KUKA KRL program: MyProgram_036().src

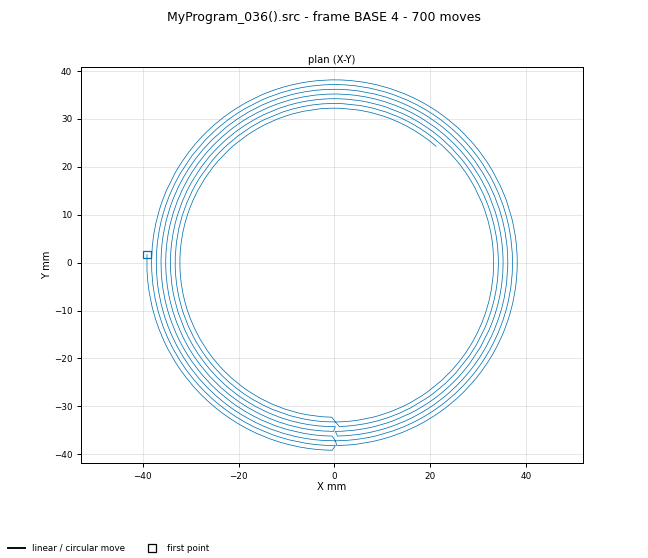
[picture p0: tool path of MyProgram_036().src in frame BASE 4, 700 of 700 moves have a stored position in this frame; points joined in program order, loops and branches not executed]
&ACCESS RVP
&REL 1
&PARAM TEMPLATE = C:\KRC\Roboter\Template\vorgabe
&PARAM EDITMASK = *
DEF MyProgram_036()
; ---- Setting reference (Base) ----
$BASE = BASE_DATA[4]

; --------------------------
; ---- Setting tool (TCP) ----
$TOOL = TOOL_DATA[3]
; --------------------------

$VEL.CP = VEL_APROX_PRINT
Startdeposition()
$VEL.CP = VEL_PRINT
LIN {X -39.1246,Y 1.7119,Z 61,A 171.6311,B 24.8459,C -2.8635,E1 24.8398,E2 -448.4299} C_DIS
LIN {X -39.1359,Y -1.4401,Z 61,A 176.0807,B 24.8477,C -2.8474,E1 24.84,E2 -452.8678} C_DIS
LIN {X -38.9837,Y -3.7356,Z 61,A 179.6269,B 24.8486,C -2.8388,E1 24.8408,E2 -456.4147} C_DIS
LIN {X -38.6887,Y -6.0708,Z 61,A -176.4142,B 24.8492,C -2.8336,E1 24.8424,E2 -460.3847} C_DIS
LIN {X -38.045,Y -9.2867,Z 61,A -172.1524,B 24.8513,C -2.8136,E1 24.8449,E2 -464.6237} C_DIS
LIN {X -37.3515,Y -11.7707,Z 61,A -167.9795,B 24.852,C -2.8066,E1 24.8483,E2 -468.8041} C_DIS
LIN {X -36.6288,Y -13.8562,Z 61,A -164.8858,B 24.8532,C -2.796,E1 24.8512,E2 -471.8898} C_DIS
LIN {X -35.5913,Y -16.3387,Z 61,A -160.9363,B 24.8543,C -2.7852,E1 24.8557,E2 -475.8352} C_DIS
LIN {X -34.7861,Y -17.9895,Z 61,A -158.0445,B 24.8548,C -2.7801,E1 24.8594,E2 -478.7304} C_DIS
LIN {X -33.1861,Y -20.7929,Z 61,A -154.2853,B 24.8572,C -2.7576,E1 24.8646,E2 -482.4552} C_DIS
LIN {X -32.2724,Y -22.1845,Z 61,A -151.2973,B 24.8572,C -2.7576,E1 24.8693,E2 -485.4579} C_DIS
LIN {X -31.1359,Y -23.754,Z 61,A -148.272,B 24.8577,C -2.7529,E1 24.8744,E2 -488.4866} C_DIS
LIN {X -29.5277,Y -25.725,Z 61,A -144.6978,B 24.8587,C -2.7428,E1 24.8808,E2 -492.0533} C_DIS
LIN {X -28.1922,Y -27.182,Z 61,A -141.5616,B 24.8591,C -2.7394,E1 24.8868,E2 -495.1951} C_DIS
LIN {X -26.3524,Y -28.9697,Z 61,A -138.0117,B 24.8601,C -2.7297,E1 24.894,E2 -498.7362} C_DIS
LIN {X -24.7345,Y -30.3624,Z 61,A -135.1218,B 24.8609,C -2.7212,E1 24.9001,E2 -501.617} C_DIS
LIN {X -23.6269,Y -31.2322,Z 61,A -132.7128,B 24.8609,C -2.7217,E1 24.9055,E2 -504.036} C_DIS
LIN {X -21.8691,Y -32.4872,Z 61,A -129.5903,B 24.8614,C -2.7162,E1 24.9127,E2 -507.1559} C_DIS
LIN {X -20.1827,Y -33.5602,Z 61,A -126.7285,B 24.8619,C -2.7112,E1 24.9195,E2 -510.0148} C_DIS
LIN {X -18.2564,Y -34.6463,Z 61,A -123.3846,B 24.8622,C -2.7083,E1 24.9277,E2 -513.3613} C_DIS
LIN {X -16.2163,Y -35.6471,Z 61,A -119.632,B 24.8621,C -2.7099,E1 24.9372,E2 -517.127} C_DIS
LIN {X -13.4921,Y -36.7645,Z 61,A -115.8847,B 24.8632,C -2.6989,E1 24.9469,E2 -520.856} C_DIS
LIN {X -11.6052,Y -37.4029,Z 61,A -112.8226,B 24.8632,C -2.6986,E1 24.955,E2 -523.9229} C_DIS
LIN {X -9.5171,Y -37.9887,Z 61,A -109.6569,B 24.8634,C -2.6966,E1 24.9636,E2 -527.0887} C_DIS
LIN {X -7.0999,Y -38.5133,Z 61,A -106.0841,B 24.8636,C -2.6946,E1 24.9733,E2 -530.6608} C_DIS
LIN {X -5.4376,Y -38.7827,Z 61,A -103.9005,B 24.8641,C -2.6903,E1 24.9794,E2 -532.8361} C_DIS
LIN {X -3.7877,Y -38.9789,Z 61,A -101.2031,B 24.8638,C -2.6936,E1 24.9869,E2 -535.5429} C_DIS
LIN {X -2.1489,Y -39.103,Z 61,A -99.0333,B 24.8641,C -2.6905,E1 24.9929,E2 -537.7062} C_DIS
LIN {X -0.4519,Y -39.16,Z 61,A -96.2889,B 24.8637,C -2.6944,E1 25.0006,E2 -540.4601} C_DIS
LIN {X -0.4519,Y -39.16,Z 61,A -96.2889,B 24.8637,C -2.6944,E1 25.0006,E2 -540.4601} C_DIS
Enddeposition()
LIN {X 0.2058,Y -38.174,Z 61,A -96.4617,B 24.8635,C -2.6964,E1 25.0001,E2 -540.2922} C_DIS
Startdeposition()
$VEL.CP = VEL_PRINT
LIN {X -1.6251,Y -38.1424,Z 61,A -99.5524,B 24.864,C -2.6916,E1 24.9915,E2 -537.1895} C_DIS
LIN {X -3.7981,Y -37.9874,Z 61,A -103.2763,B 24.8645,C -2.686,E1 24.9811,E2 -533.4505} C_DIS
LIN {X -5.7354,Y -37.7438,Z 61,A -106.8998,B 24.8653,C -2.6781,E1 24.971,E2 -529.8052} C_DIS
LIN {X -9.3911,Y -37.0041,Z 61,A -111.3776,B 24.8637,C -2.6944,E1 24.9589,E2 -525.3603} C_DIS
LIN {X -11.7237,Y -36.3323,Z 61,A -114.7703,B 24.8631,C -2.6999,E1 24.9498,E2 -521.975} C_DIS
LIN {X -12.9207,Y -35.9244,Z 61,A -117.5141,B 24.864,C -2.6915,E1 24.9426,E2 -519.2057} C_DIS
LIN {X -16.5245,Y -34.4154,Z 61,A -122.843,B 24.8627,C -2.7039,E1 24.929,E2 -513.8936} C_DIS
LIN {X -18.8039,Y -33.2249,Z 61,A -126.9062,B 24.8624,C -2.7066,E1 24.919,E2 -509.8253} C_DIS
LIN {X -20.5168,Y -32.1953,Z 61,A -129.5033,B 24.8615,C -2.7154,E1 24.9129,E2 -507.2414} C_DIS
LIN {X -21.5761,Y -31.496,Z 61,A -131.5541,B 24.8614,C -2.7168,E1 24.9081,E2 -505.1869} C_DIS
LIN {X -22.9175,Y -30.5331,Z 61,A -134.0934,B 24.861,C -2.7203,E1 24.9024,E2 -502.647} C_DIS
LIN {X -24.5041,Y -29.2754,Z 61,A -136.9789,B 24.8603,C -2.7274,E1 24.8962,E2 -499.7676} C_DIS
LIN {X -25.6498,Y -28.2775,Z 61,A -139.37,B 24.86,C -2.7306,E1 24.8912,E2 -497.3745} C_DIS
LIN {X -26.978,Y -27.0123,Z 61,A -142.0686,B 24.8593,C -2.7367,E1 24.8858,E2 -494.6794} C_DIS
LIN {X -28.1489,Y -25.79,Z 61,A -144.6778,B 24.8588,C -2.7414,E1 24.8808,E2 -492.07} C_DIS
LIN {X -29.33,Y -24.4382,Z 61,A -147.3487,B 24.8582,C -2.7477,E1 24.876,E2 -489.4019} C_DIS
LIN {X -30.4284,Y -23.0568,Z 61,A -149.8973,B 24.8575,C -2.7549,E1 24.8716,E2 -486.8585} C_DIS
LIN {X -31.2137,Y -21.9816,Z 61,A -152.4219,B 24.8575,C -2.7544,E1 24.8675,E2 -484.3202} C_DIS
LIN {X -32.4672,Y -20.0846,Z 61,A -155.857,B 24.8566,C -2.7627,E1 24.8623,E2 -480.8877} C_DIS
LIN {X -33.8432,Y -17.6674,Z 61,A -159.701,B 24.8551,C -2.777,E1 24.8572,E2 -477.0576} C_DIS
LIN {X -34.9349,Y -15.3963,Z 61,A -163.7856,B 24.8544,C -2.7844,E1 24.8524,E2 -472.9685} C_DIS
LIN {X -35.7598,Y -13.369,Z 61,A -167.3157,B 24.8536,C -2.7914,E1 24.8488,E2 -469.4352} C_DIS
LIN {X -36.7499,Y -10.3404,Z 61,A -171.6234,B 24.8517,C -2.81,E1 24.8453,E2 -465.1472} C_DIS
LIN {X -37.4441,Y -7.4482,Z 61,A -177.1229,B 24.8513,C -2.8136,E1 24.842,E2 -459.6239} C_DIS
LIN {X -37.8937,Y -4.6464,Z 61,A 179.0092,B 24.8495,C -2.8303,E1 24.8406,E2 -455.7729} C_DIS
LIN {X -38.1362,Y -1.7679,Z 61,A 175.1413,B 24.8476,C -2.8482,E1 24.8399,E2 -451.9246} C_DIS
LIN {X -38.1731,Y 0.5611,Z 61,A 170.9288,B 24.8471,C -2.8524,E1 24.8399,E2 -447.6968} C_DIS
LIN {X -38.0202,Y 3.4564,Z 61,A 167.0952,B 24.8451,C -2.8709,E1 24.8407,E2 -443.8844} C_DIS
LIN {X -37.7315,Y 5.815,Z 61,A 163.5178,B 24.844,C -2.8819,E1 24.842,E2 -440.3121} C_DIS
LIN {X -37.28,Y 8.2277,Z 61,A 159.4344,B 24.8431,C -2.8896,E1 24.8444,E2 -436.2229} C_DIS
LIN {X -36.5358,Y 11.0755,Z 61,A 155.6693,B 24.841,C -2.9093,E1 24.8472,E2 -432.4832} C_DIS
LIN {X -35.9396,Y 12.8788,Z 61,A 152.4915,B 24.8404,C -2.9148,E1 24.85,E2 -429.3004} C_DIS
LIN {X -35.1002,Y 15.0163,Z 61,A 148.4463,B 24.8399,C -2.9193,E1 24.8544,E2 -425.2436} C_DIS
LIN {X -33.2218,Y 18.8107,Z 61,A 143.1464,B 24.8367,C -2.9477,E1 24.8611,E2 -419.9833} C_DIS
LIN {X -32.099,Y 20.6674,Z 61,A 138.9421,B 24.8367,C -2.9475,E1 24.8674,E2 -415.757} C_DIS
LIN {X -30.4008,Y 23.0936,Z 61,A 134.5485,B 24.8354,C -2.9597,E1 24.8746,E2 -411.3713} C_DIS
LIN {X -28.9431,Y 24.896,Z 61,A 131.6927,B 24.8337,C -2.9747,E1 24.8797,E2 -408.5383} C_DIS
LIN {X -27.8474,Y 26.1152,Z 61,A 129.0954,B 24.8332,C -2.9793,E1 24.8846,E2 -405.9406} C_DIS
LIN {X -26.5489,Y 27.4343,Z 61,A 126.228,B 24.8326,C -2.9849,E1 24.8902,E2 -403.0744} C_DIS
LIN {X -24.9689,Y 28.8796,Z 61,A 122.2932,B 24.8326,C -2.9846,E1 24.8985,E2 -399.1234} C_DIS
LIN {X -22.971,Y 30.4929,Z 61,A 119.3529,B 24.8306,C -3.0021,E1 24.9049,E2 -396.2141} C_DIS
LIN {X -20.951,Y 31.9146,Z 61,A 114.7776,B 24.8308,C -3,E1 24.9155,E2 -391.6186} C_DIS
LIN {X -18.3987,Y 33.4508,Z 61,A 110.4355,B 24.8298,C -3.0091,E1 24.9261,E2 -387.2853} C_DIS
LIN {X -15.4253,Y 34.9224,Z 61,A 106.0547,B 24.8282,C -3.0232,E1 24.937,E2 -382.9271} C_DIS
LIN {X -13.9822,Y 35.5244,Z 61,A 103.7511,B 24.8278,C -3.0269,E1 24.943,E2 -380.6271} C_DIS
LIN {X -12.4032,Y 36.1066,Z 61,A 101.0674,B 24.8276,C -3.0282,E1 24.9501,E2 -377.9413} C_DIS
LIN {X -10.6068,Y 36.6745,Z 61,A 98.1852,B 24.8274,C -3.0307,E1 24.9578,E2 -375.06} C_DIS
LIN {X -8.7748,Y 37.1544,Z 61,A 94.9865,B 24.8275,C -3.0292,E1 24.9665,E2 -371.8533} C_DIS
LIN {X -6.2361,Y 37.6642,Z 61,A 91.3939,B 24.8268,C -3.0356,E1 24.9763,E2 -368.2722} C_DIS
LIN {X -3.4721,Y 38.0188,Z 61,A 86.7795,B 24.8271,C -3.0326,E1 24.9891,E2 -363.648} C_DIS
LIN {X -0.5874,Y 38.1726,Z 61,A 82.9526,B 24.8263,C -3.0402,E1 24.9997,E2 -359.8384} C_DIS
LIN {X 1.5062,Y 38.1473,Z 61,A 79.9793,B 24.826,C -3.0427,E1 25.008,E2 -356.8715} C_DIS
LIN {X 3.3481,Y 38.03,Z 61,A 76.4399,B 24.8271,C -3.0328,E1 25.0179,E2 -353.3105} C_DIS
LIN {X 6.3001,Y 37.6535,Z 61,A 72.8307,B 24.826,C -3.0427,E1 25.0278,E2 -349.728} C_DIS
LIN {X 8.7875,Y 37.1523,Z 61,A 68.6153,B 24.8268,C -3.0356,E1 25.0394,E2 -345.5011} C_DIS
LIN {X 11.5673,Y 36.3827,Z 61,A 63.6954,B 24.828,C -3.0247,E1 25.0526,E2 -340.564} C_DIS
LIN {X 14.6024,Y 35.2747,Z 61,A 59.3124,B 24.8278,C -3.0264,E1 25.064,E2 -336.1945} C_DIS
LIN {X 16.5716,Y 34.3928,Z 61,A 56.4111,B 24.8278,C -3.0273,E1 25.0713,E2 -333.3029} C_DIS
LIN {X 18.0246,Y 33.6545,Z 61,A 54.01,B 24.828,C -3.0248,E1 25.0772,E2 -330.9025} C_DIS
LIN {X 19.4873,Y 32.8288,Z 61,A 51.7271,B 24.828,C -3.0247,E1 25.0827,E2 -328.6262} C_DIS
LIN {X 20.561,Y 32.1673,Z 61,A 49.7273,B 24.8285,C -3.0203,E1 25.0875,E2 -326.6224} C_DIS
LIN {X 21.7389,Y 31.3832,Z 61,A 47.3022,B 24.8294,C -3.0126,E1 25.0931,E2 -324.1873} C_DIS
LIN {X 23.4845,Y 30.0999,Z 61,A 43.8809,B 24.8303,C -3.0045,E1 25.1007,E2 -320.7592} C_DIS
LIN {X 25.6796,Y 28.2502,Z 61,A 40.0705,B 24.8304,C -3.0036,E1 25.1087,E2 -316.9615} C_DIS
LIN {X 26.6253,Y 27.3604,Z 61,A 37.5195,B 24.8319,C -2.9908,E1 25.1139,E2 -314.3909} C_DIS
LIN {X 28.6369,Y 25.2476,Z 61,A 33.4573,B 24.8324,C -2.986,E1 25.1215,E2 -310.3351} C_DIS
LIN {X 30.1948,Y 23.3613,Z 61,A 29.8375,B 24.8333,C -2.9783,E1 25.1279,E2 -306.7139} C_DIS
LIN {X 31.7933,Y 21.1349,Z 61,A 25.3674,B 24.835,C -2.9628,E1 25.135,E2 -302.229} C_DIS
LIN {X 32.9335,Y 19.3101,Z 61,A 22.073,B 24.8361,C -2.9534,E1 25.1397,E2 -298.9294} C_DIS
LIN {X 34.6066,Y 16.1204,Z 61,A 17.177,B 24.8368,C -2.9466,E1 25.1458,E2 -294.0434} C_DIS
LIN {X 35.5024,Y 14.0382,Z 61,A 13.9544,B 24.8376,C -2.9399,E1 25.1493,E2 -290.8225} C_DIS
LIN {X 35.9963,Y 12.7183,Z 61,A 11.2382,B 24.8393,C -2.9244,E1 25.1518,E2 -288.085} C_DIS
LIN {X 37.0311,Y 9.2859,Z 61,A 6.2712,B 24.8403,C -2.915,E1 25.1556,E2 -283.124} C_DIS
LIN {X 37.3917,Y 7.7034,Z 61,A 3.9387,B 24.841,C -2.9092,E1 25.1569,E2 -280.7916} C_DIS
LIN {X 37.7634,Y 5.6075,Z 61,A 0.7109,B 24.8421,C -2.8989,E1 25.1584,E2 -277.5584} C_DIS
LIN {X 37.9807,Y 3.8676,Z 61,A -1.8164,B 24.8428,C -2.8925,E1 25.1592,E2 -275.0307} C_DIS
LIN {X 38.1283,Y 1.9349,Z 61,A -4.6115,B 24.8436,C -2.8852,E1 25.1597,E2 -272.235} C_DIS
LIN {X 38.1752,Y 0.4157,Z 61,A -6.7829,B 24.8442,C -2.8798,E1 25.1597,E2 -270.0638} C_DIS
LIN {X 38.1514,Y -1.4106,Z 61,A -9.8132,B 24.8456,C -2.8666,E1 25.1596,E2 -267.0204} C_DIS
LIN {X 38.0292,Y -3.3592,Z 61,A -12.4507,B 24.8461,C -2.8621,E1 25.159,E2 -264.3877} C_DIS
LIN {X 37.7783,Y -5.5026,Z 61,A -15.9673,B 24.8477,C -2.8475,E1 25.1577,E2 -260.8574} C_DIS
LIN {X 37.249,Y -8.3648,Z 61,A -20.7885,B 24.8499,C -2.8268,E1 25.155,E2 -256.0153} C_DIS
LIN {X 36.6348,Y -10.7419,Z 61,A -23.6115,B 24.8496,C -2.8291,E1 25.1529,E2 -253.2138} C_DIS
LIN {X 36.227,Y -12.0447,Z 61,A -25.7983,B 24.8505,C -2.8206,E1 25.151,E2 -251.0194} C_DIS
LIN {X 35.4552,Y -14.1583,Z 61,A -28.9661,B 24.8513,C -2.8138,E1 25.1479,E2 -247.8531} C_DIS
LIN {X 34.7913,Y -15.7177,Z 61,A -31.8323,B 24.8526,C -2.8012,E1 25.1447,E2 -244.9727} C_DIS
LIN {X 33.868,Y -17.6204,Z 61,A -34.7421,B 24.8531,C -2.7961,E1 25.141,E2 -242.0665} C_DIS
LIN {X 33.0339,Y -19.1379,Z 61,A -37.4369,B 24.8541,C -2.7872,E1 25.1373,E2 -239.3646} C_DIS
LIN {X 32.2579,Y -20.4193,Z 61,A -40.0322,B 24.8553,C -2.7756,E1 25.1334,E2 -236.755} C_DIS
LIN {X 30.6847,Y -22.715,Z 61,A -43.7394,B 24.8557,C -2.7717,E1 25.1275,E2 -233.0564} C_DIS
LIN {X 29.6057,Y -24.1037,Z 61,A -46.2431,B 24.8562,C -2.7669,E1 25.1231,E2 -230.5532} C_DIS
LIN {X 28.6953,Y -25.1808,Z 61,A -48.7794,B 24.8574,C -2.7552,E1 25.1185,E2 -228.0005} C_DIS
LIN {X 26.8749,Y -27.1148,Z 61,A -52.4982,B 24.858,C -2.7496,E1 25.1112,E2 -224.2846} C_DIS
LIN {X 25.4921,Y -28.4183,Z 61,A -55.5822,B 24.859,C -2.7396,E1 25.1049,E2 -221.1894} C_DIS
LIN {X 23.4955,Y -30.091,Z 61,A -59.0641,B 24.8592,C -2.7376,E1 25.0974,E2 -217.7159} C_DIS
LIN {X 22.3346,Y -30.9625,Z 61,A -61.3187,B 24.8598,C -2.732,E1 25.0923,E2 -215.4561} C_DIS
LIN {X 20.9688,Y -31.9029,Z 61,A -64.0449,B 24.8607,C -2.7237,E1 25.0859,E2 -212.7194} C_DIS
LIN {X 18.8062,Y -33.2233,Z 61,A -67.5439,B 24.8609,C -2.7213,E1 25.0775,E2 -209.2255} C_DIS
LIN {X 17.0992,Y -34.1339,Z 61,A -70.8441,B 24.862,C -2.7109,E1 25.0693,E2 -205.9096} C_DIS
LIN {X 14.4634,Y -35.3313,Z 61,A -75.3242,B 24.8628,C -2.7027,E1 25.0578,E2 -201.4207} C_DIS
LIN {X 11.9187,Y -36.2692,Z 61,A -78.7995,B 24.8625,C -2.7059,E1 25.0487,E2 -197.9601} C_DIS
LIN {X 9.9784,Y -36.8499,Z 61,A -82.0849,B 24.8632,C -2.6992,E1 25.0398,E2 -194.6643} C_DIS
LIN {X 7.9305,Y -37.3437,Z 61,A -85.4763,B 24.8638,C -2.6932,E1 25.0306,E2 -191.2633} C_DIS
LIN {X 4.7796,Y -37.8768,Z 61,A -89.56,B 24.8632,C -2.6994,E1 25.0194,E2 -187.1982} C_DIS
LIN {X 2.7394,Y -38.0789,Z 61,A -93.3905,B 24.8643,C -2.6879,E1 25.0086,E2 -183.3425} C_DIS
LIN {X 0.4929,Y -38.1744,Z 61,A -96.4487,B 24.864,C -2.6909,E1 25.0001,E2 -180.2922} C_DIS
LIN {X 0.4929,Y -38.1744,Z 61,A -96.4487,B 24.864,C -2.6909,E1 25.0001,E2 -180.2922} C_DIS
Enddeposition()
LIN {X 0.2169,Y -37.1885,Z 61,A -97.0627,B 24.8625,C -2.7057,E1 24.9985,E2 -179.7131} C_DIS
Startdeposition()
$VEL.CP = VEL_PRINT
LIN {X 2.3849,Y -37.1156,Z 61,A -91.3777,B 24.8593,C -2.7372,E1 25.0146,E2 -185.4716} C_DIS
LIN {X 4.4565,Y -36.9242,Z 61,A -88.3914,B 24.8593,C -2.7362,E1 25.0228,E2 -188.4532} C_DIS
LIN {X 7.033,Y -36.5207,Z 61,A -84.9258,B 24.8598,C -2.7317,E1 25.0323,E2 -191.9046} C_DIS
LIN {X 8.6705,Y -36.1675,Z 61,A -81.6512,B 24.8586,C -2.7437,E1 25.0413,E2 -195.203} C_DIS
LIN {X 12.3086,Y -35.0962,Z 61,A -76.6912,B 24.8592,C -2.7381,E1 25.0544,E2 -200.1407} C_DIS
LIN {X 14.4746,Y -34.2597,Z 61,A -72.4913,B 24.8578,C -2.7518,E1 25.0654,E2 -204.3637} C_DIS
LIN {X 16.5626,Y -33.3005,Z 61,A -69.4009,B 24.8578,C -2.7509,E1 25.0731,E2 -207.4438} C_DIS
LIN {X 18.2017,Y -32.4337,Z 61,A -66.4981,B 24.8573,C -2.7564,E1 25.0803,E2 -210.3514} C_DIS
LIN {X 19.8235,Y -31.4689,Z 61,A -63.5956,B 24.8567,C -2.7617,E1 25.0872,E2 -213.2571} C_DIS
LIN {X 21.6468,Y -30.2433,Z 61,A -60.2084,B 24.856,C -2.7684,E1 25.095,E2 -216.6487} C_DIS
LIN {X 23.1585,Y -29.1023,Z 61,A -57.1197,B 24.8551,C -2.777,E1 25.1018,E2 -219.7466} C_DIS
LIN {X 25.1549,Y -27.3948,Z 61,A -53.3687,B 24.8547,C -2.7817,E1 25.1096,E2 -223.4936} C_DIS
LIN {X 26.8232,Y -25.7636,Z 61,A -49.4807,B 24.8533,C -2.7947,E1 25.1173,E2 -227.3959} C_DIS
LIN {X 28.2812,Y -24.154,Z 61,A -46.3833,B 24.8528,C -2.7992,E1 25.123,E2 -230.4902} C_DIS
LIN {X 29.3197,Y -22.8833,Z 61,A -44.0555,B 24.8524,C -2.8027,E1 25.1271,E2 -232.8153} C_DIS
LIN {X 30.3514,Y -21.4954,Z 61,A -41.1551,B 24.8513,C -2.8135,E1 25.1318,E2 -235.7271} C_DIS
LIN {X 31.3778,Y -19.9674,Z 61,A -38.5235,B 24.8508,C -2.8181,E1 25.1359,E2 -238.3565} C_DIS
LIN {X 32.3405,Y -18.3676,Z 61,A -35.4557,B 24.8496,C -2.8291,E1 25.1402,E2 -241.4347} C_DIS
LIN {X 33.2135,Y -16.7376,Z 61,A -32.7932,B 24.8491,C -2.8344,E1 25.1436,E2 -244.0957} C_DIS
LIN {X 34.1529,Y -14.7256,Z 61,A -29.1477,B 24.8476,C -2.8481,E1 25.1478,E2 -247.7536} C_DIS
LIN {X 35.1839,Y -12.0569,Z 61,A -24.4656,B 24.8457,C -2.8657,E1 25.1523,E2 -252.4513} C_DIS
LIN {X 35.8338,Y -9.9607,Z 61,A -21.81,B 24.8458,C -2.8646,E1 25.1544,E2 -255.089} C_DIS
LIN {X 36.3501,Y -7.8679,Z 61,A -18.0003,B 24.8439,C -2.8826,E1 25.1568,E2 -258.9194} C_DIS
LIN {X 36.86,Y -4.9553,Z 61,A -13.15,B 24.8418,C -2.9016,E1 25.1588,E2 -263.786} C_DIS
LIN {X 37.1169,Y -2.3657,Z 61,A -9.6045,B 24.8412,C -2.9067,E1 25.1596,E2 -267.3227} C_DIS
LIN {X 37.1908,Y -0.1047,Z 61,A -6.4021,B 24.8405,C -2.9132,E1 25.1598,E2 -270.5213} C_DIS
LIN {X 37.1307,Y 2.1343,Z 61,A -2.5235,B 24.8386,C -2.9307,E1 25.1593,E2 -274.4183} C_DIS
LIN {X 36.8227,Y 5.2278,Z 61,A 2.0615,B 24.8373,C -2.9422,E1 25.1578,E2 -279.0035} C_DIS
LIN {X 36.3889,Y 7.6901,Z 61,A 5.9718,B 24.8359,C -2.9548,E1 25.1557,E2 -282.9208} C_DIS
LIN {X 35.9015,Y 9.7122,Z 61,A 9.0106,B 24.8351,C -2.9618,E1 25.1536,E2 -285.9585} C_DIS
LIN {X 35.2316,Y 11.9155,Z 61,A 12.6038,B 24.8339,C -2.9728,E1 25.1505,E2 -289.5575} C_DIS
LIN {X 34.2434,Y 14.5133,Z 61,A 16.4426,B 24.8333,C -2.9781,E1 25.1466,E2 -293.3875} C_DIS
LIN {X 33.3854,Y 16.3914,Z 61,A 19.7505,B 24.8321,C -2.9888,E1 25.1426,E2 -296.7028} C_DIS
LIN {X 32.6017,Y 17.8994,Z 61,A 22.5447,B 24.831,C -2.9984,E1 25.1389,E2 -299.5052} C_DIS
LIN {X 31.0625,Y 20.454,Z 61,A 27.4269,B 24.8292,C -3.0145,E1 25.1316,E2 -304.4009} C_DIS
LIN {X 29.9798,Y 22.0103,Z 61,A 30.226,B 24.8286,C -3.0197,E1 25.1271,E2 -307.1988} C_DIS
LIN {X 28.5043,Y 23.8906,Z 61,A 33.4788,B 24.8284,C -3.0217,E1 25.1213,E2 -310.4413} C_DIS
LIN {X 27.2141,Y 25.3508,Z 61,A 36.673,B 24.8273,C -3.0311,E1 25.1153,E2 -313.6436} C_DIS
LIN {X 25.9716,Y 26.6224,Z 61,A 39.0983,B 24.8272,C -3.0322,E1 25.1106,E2 -316.0611} C_DIS
LIN {X 24.9231,Y 27.6063,Z 61,A 41.2999,B 24.8267,C -3.0364,E1 25.106,E2 -318.2637} C_DIS
LIN {X 23.5916,Y 28.7528,Z 61,A 44.243,B 24.8257,C -3.0448,E1 25.0997,E2 -321.2155} C_DIS
LIN {X 22.1541,Y 29.8745,Z 61,A 46.8689,B 24.8255,C -3.047,E1 25.0939,E2 -323.8372} C_DIS
LIN {X 20.6785,Y 30.9141,Z 61,A 49.7704,B 24.8248,C -3.0532,E1 25.0872,E2 -326.7435} C_DIS
LIN {X 19.1363,Y 31.8912,Z 61,A 52.5284,B 24.8244,C -3.0566,E1 25.0806,E2 -329.5008} C_DIS
LIN {X 17.3082,Y 32.9185,Z 61,A 55.5259,B 24.8242,C -3.0577,E1 25.0733,E2 -332.4922} C_DIS
LIN {X 15.2138,Y 33.938,Z 61,A 60.0822,B 24.8222,C -3.0751,E1 25.0617,E2 -337.0782} C_DIS
LIN {X 12.2259,Y 35.125,Z 61,A 64.1899,B 24.823,C -3.0681,E1 25.051,E2 -341.1607} C_DIS
LIN {X 10.4794,Y 35.6852,Z 61,A 67.3895,B 24.8222,C -3.0751,E1 25.0424,E2 -344.3713} C_DIS
LIN {X 7.3773,Y 36.4531,Z 61,A 72.7453,B 24.8213,C -3.0833,E1 25.0278,E2 -349.7392} C_DIS
LIN {X 4.2796,Y 36.9449,Z 61,A 76.9883,B 24.822,C -3.0768,E1 25.0161,E2 -353.9632} C_DIS
LIN {X 2.0522,Y 37.1353,Z 61,A 80.0907,B 24.8225,C -3.0726,E1 25.0075,E2 -357.0541} C_DIS
LIN {X 0.5284,Y 37.1878,Z 61,A 82.3741,B 24.8226,C -3.0715,E1 25.0012,E2 -359.3346} C_DIS
LIN {X -0.7909,Y 37.1837,Z 61,A 84.5758,B 24.8225,C -3.0731,E1 24.995,E2 -361.5402} C_DIS
LIN {X -2.4496,Y 37.1112,Z 61,A 87.4123,B 24.8222,C -3.0756,E1 24.9871,E2 -364.3833} C_DIS
LIN {X -4.8206,Y 36.8781,Z 61,A 91.0006,B 24.8225,C -3.0726,E1 24.9771,E2 -367.9668} C_DIS
LIN {X -7.0528,Y 36.5171,Z 61,A 94.5567,B 24.8227,C -3.0709,E1 24.9674,E2 -371.5224} C_DIS
LIN {X -8.7501,Y 36.1478,Z 61,A 97.2717,B 24.8229,C -3.0689,E1 24.96,E2 -374.2364} C_DIS
LIN {X -11.2846,Y 35.4391,Z 61,A 101.615,B 24.8231,C -3.0678,E1 24.9484,E2 -378.5844} C_DIS
LIN {X -13.9275,Y 34.4856,Z 61,A 105.2739,B 24.8246,C -3.0547,E1 24.9389,E2 -382.2197} C_DIS
LIN {X -15.2481,Y 33.9225,Z 61,A 108.3606,B 24.8238,C -3.0612,E1 24.9309,E2 -385.3294} C_DIS
LIN {X -18.6585,Y 32.1733,Z 61,A 113.2512,B 24.8262,C -3.0405,E1 24.919,E2 -390.1841} C_DIS
LIN {X -20.4585,Y 31.0595,Z 61,A 117.3806,B 24.8259,C -3.0437,E1 24.9092,E2 -394.3345} C_DIS
LIN {X -22.133,Y 29.8893,Z 61,A 120.2372,B 24.8269,C -3.0344,E1 24.9028,E2 -397.1787} C_DIS
LIN {X -24.6646,Y 27.8376,Z 61,A 125.9041,B 24.8274,C -3.0302,E1 24.8907,E2 -402.8576} C_DIS
LIN {X -26.9264,Y 25.6557,Z 61,A 130.8491,B 24.8286,C -3.0198,E1 24.881,E2 -407.7989} C_DIS
LIN {X -29.7226,Y 22.3565,Z 61,A 137.7372,B 24.8303,C -3.005,E1 24.8691,E2 -414.6837} C_DIS
LIN {X -32.2026,Y 18.6075,Z 61,A 143.445,B 24.8338,C -2.9739,E1 24.8606,E2 -420.3462} C_DIS
LIN {X -33.3982,Y 16.3649,Z 61,A 148.1652,B 24.8342,C -2.9705,E1 24.8546,E2 -425.0834} C_DIS
LIN {X -34.4531,Y 14.0081,Z 61,A 151.5876,B 24.8361,C -2.9534,E1 24.8509,E2 -428.4838} C_DIS
LIN {X -35.1923,Y 12.0319,Z 61,A 155.0714,B 24.8369,C -2.9458,E1 24.8476,E2 -431.9693} C_DIS
LIN {X -35.7811,Y 10.1465,Z 61,A 157.8531,B 24.8382,C -2.934,E1 24.8454,E2 -434.7388} C_DIS
LIN {X -36.1965,Y 8.5471,Z 61,A 160.5632,B 24.8389,C -2.9277,E1 24.8436,E2 -437.4497} C_DIS
LIN {X -36.5512,Y 6.8758,Z 61,A 163.298,B 24.8397,C -2.9205,E1 24.8421,E2 -440.1835} C_DIS
LIN {X -36.9253,Y 4.447,Z 61,A 166.8818,B 24.8412,C -2.9068,E1 24.8407,E2 -443.7557} C_DIS
LIN {X -37.1012,Y 2.5983,Z 61,A 169.982,B 24.842,C -2.9001,E1 24.84,E2 -446.8585} C_DIS
LIN {X -37.1853,Y 0.7016,Z 61,A 173.1958,B 24.8427,C -2.8937,E1 24.8398,E2 -450.0764} C_DIS
LIN {X -37.1328,Y -2.097,Z 61,A 176.9044,B 24.8447,C -2.8745,E1 24.8401,E2 -453.7615} C_DIS
LIN {X -36.9128,Y -4.553,Z 61,A -179.4157,B 24.8461,C -2.8617,E1 24.8411,E2 -457.4326} C_DIS
LIN {X -36.7209,Y -5.9031,Z 61,A -176.5103,B 24.8461,C -2.8629,E1 24.8424,E2 -460.3582} C_DIS
LIN {X -36.1431,Y -8.7705,Z 61,A -172.3751,B 24.8479,C -2.8458,E1 24.8448,E2 -464.4768} C_DIS
LIN {X -35.4628,Y -11.2093,Z 61,A -168.0498,B 24.8486,C -2.8384,E1 24.8483,E2 -468.8095} C_DIS
LIN {X -34.7074,Y -13.3653,Z 61,A -164.8886,B 24.8501,C -2.8249,E1 24.8513,E2 -471.9561} C_DIS
LIN {X -33.9717,Y -15.139,Z 61,A -161.8008,B 24.8508,C -2.8179,E1 24.8547,E2 -475.0443} C_DIS
LIN {X -32.8997,Y -17.3451,Z 61,A -157.9791,B 24.8519,C -2.8082,E1 24.8595,E2 -478.8631} C_DIS
LIN {X -31.7468,Y -19.3748,Z 61,A -154.4433,B 24.8529,C -2.7983,E1 24.8645,E2 -482.3937} C_DIS
LIN {X -30.6809,Y -21.023,Z 61,A -151.487,B 24.8538,C -2.7901,E1 24.8691,E2 -485.3451} C_DIS
LIN {X -29.7205,Y -22.3592,Z 61,A -148.9048,B 24.8544,C -2.7845,E1 24.8734,E2 -487.9265} C_DIS
LIN {X -28.2607,Y -24.1781,Z 61,A -145.0918,B 24.855,C -2.7786,E1 24.8802,E2 -491.7431} C_DIS
LIN {X -26.6562,Y -25.9367,Z 61,A -141.3564,B 24.8557,C -2.7716,E1 24.8873,E2 -495.4779} C_DIS
LIN {X -24.947,Y -27.5849,Z 61,A -137.9331,B 24.8567,C -2.7618,E1 24.8943,E2 -498.8918} C_DIS
LIN {X -23.2181,Y -29.0549,Z 61,A -134.1761,B 24.8571,C -2.7583,E1 24.9024,E2 -502.6548} C_DIS
LIN {X -21.6219,Y -30.2611,Z 61,A -131.4017,B 24.858,C -2.7498,E1 24.9086,E2 -505.4185} C_DIS
LIN {X -20.4307,Y -31.0777,Z 61,A -129.2334,B 24.8584,C -2.7457,E1 24.9137,E2 -507.5843} C_DIS
LIN {X -19.2213,Y -31.8401,Z 61,A -126.5407,B 24.8582,C -2.7481,E1 24.9201,E2 -510.291} C_DIS
LIN {X -16.6353,Y -33.2645,Z 61,A -122.4847,B 24.8593,C -2.7366,E1 24.9301,E2 -514.3311} C_DIS
LIN {X -14.9445,Y -34.0575,Z 61,A -119.3732,B 24.8593,C -2.7362,E1 24.938,E2 -517.4491} C_DIS
LIN {X -13.2562,Y -34.7493,Z 61,A -116.4906,B 24.8596,C -2.7345,E1 24.9455,E2 -520.3337} C_DIS
LIN {X -10.6338,Y -35.6394,Z 61,A -111.8564,B 24.8594,C -2.7357,E1 24.9579,E2 -524.9794} C_DIS
LIN {X -8.1583,Y -36.2868,Z 61,A -108.0068,B 24.8598,C -2.7326,E1 24.9683,E2 -528.8266} C_DIS
LIN {X -5.9808,Y -36.7082,Z 61,A -105.078,B 24.8605,C -2.7254,E1 24.9763,E2 -531.7413} C_DIS
LIN {X -4.2976,Y -36.9427,Z 61,A -102.3196,B 24.8604,C -2.7268,E1 24.984,E2 -534.5049} C_DIS
LIN {X -2.4007,Y -37.1145,Z 61,A -99.2123,B 24.8601,C -2.729,E1 24.9927,E2 -537.6186} C_DIS
LIN {X 0.2169,Y -37.1885,Z 61,A -97.0625,B 24.8625,C -2.7056,E1 24.9985,E2 -539.7131} C_DIS
Enddeposition()
LIN {X 0.2169,Y -37.1885,Z 61,A -97.0625,B 24.8625,C -2.7056,E1 24.9985,E2 -539.7131} C_DIS
Startdeposition()
$VEL.CP = VEL_PRINT
LIN {X -0.4707,Y -36.2042,Z 61,A -97.8735,B 24.8604,C -2.7261,E1 24.9964,E2 -538.9508} C_DIS
LIN {X -2.2002,Y -36.1406,Z 61,A -100.9136,B 24.8608,C -2.7222,E1 24.9879,E2 -535.9007} C_DIS
LIN {X -4.2357,Y -35.9583,Z 61,A -103.7817,B 24.8603,C -2.7269,E1 24.9799,E2 -533.0422} C_DIS
LIN {X -6.2267,Y -35.6673,Z 61,A -107.5775,B 24.861,C -2.7206,E1 24.9694,E2 -529.2278} C_DIS
LIN {X -9.7757,Y -34.8624,Z 61,A -113.6647,B 24.861,C -2.72,E1 24.9529,E2 -523.1305} C_DIS
LIN {X -12.2444,Y -34.0737,Z 61,A -117.5654,B 24.8605,C -2.7256,E1 24.9426,E2 -519.2356} C_DIS
LIN {X -15.2233,Y -32.8511,Z 61,A -122.0554,B 24.8593,C -2.7375,E1 24.9312,E2 -514.7634} C_DIS
LIN {X -16.8727,Y -32.0352,Z 61,A -124.9767,B 24.8589,C -2.7409,E1 24.9239,E2 -511.8425} C_DIS
LIN {X -18.4966,Y -31.126,Z 61,A -127.9408,B 24.8585,C -2.7447,E1 24.9167,E2 -508.8786} C_DIS
LIN {X -20.4252,Y -29.8961,Z 61,A -131.4292,B 24.8578,C -2.7516,E1 24.9086,E2 -505.3953} C_DIS
LIN {X -21.4978,Y -29.1343,Z 61,A -134.1715,B 24.8581,C -2.7483,E1 24.9024,E2 -502.6354} C_DIS
LIN {X -24.0379,Y -27.0766,Z 61,A -138.6657,B 24.8564,C -2.7647,E1 24.8928,E2 -498.1631} C_DIS
LIN {X -25.7628,Y -25.4399,Z 61,A -143.0238,B 24.8563,C -2.7664,E1 24.884,E2 -493.7909} C_DIS
LIN {X -27.7429,Y -23.2639,Z 61,A -148.1784,B 24.8557,C -2.7719,E1 24.8746,E2 -488.6261} C_DIS
LIN {X -29.7511,Y -20.6353,Z 61,A -152.6709,B 24.8536,C -2.7915,E1 24.8672,E2 -484.1587} C_DIS
LIN {X -30.6815,Y -19.2247,Z 61,A -155.06,B 24.8526,C -2.8009,E1 24.8636,E2 -481.78} C_DIS
LIN {X -31.4901,Y -17.8705,Z 61,A -157.8463,B 24.8522,C -2.8046,E1 24.8597,E2 -478.9882} C_DIS
LIN {X -32.328,Y -16.305,Z 61,A -160.6897,B 24.8515,C -2.8118,E1 24.8561,E2 -476.1468} C_DIS
LIN {X -33.1545,Y -14.5509,Z 61,A -164.2092,B 24.851,C -2.8162,E1 24.852,E2 -472.6184} C_DIS
LIN {X -34.2139,Y -11.8478,Z 61,A -168.39,B 24.8492,C -2.833,E1 24.848,E2 -468.4544} C_DIS
LIN {X -34.8201,Y -9.925,Z 61,A -171.588,B 24.8482,C -2.8423,E1 24.8454,E2 -465.2602} C_DIS
LIN {X -35.3212,Y -7.9617,Z 61,A -174.6284,B 24.847,C -2.8534,E1 24.8434,E2 -462.2284} C_DIS
LIN {X -35.7955,Y -5.4435,Z 61,A -178.5646,B 24.8456,C -2.8668,E1 24.8414,E2 -458.301} C_DIS
LIN {X -36.0199,Y -3.6754,Z 61,A 178.3273,B 24.8449,C -2.8729,E1 24.8404,E2 -455.189} C_DIS
LIN {X -36.1515,Y -2.0022,Z 61,A 175.4227,B 24.8443,C -2.879,E1 24.8399,E2 -452.2813} C_DIS
LIN {X -36.2039,Y 0.494,Z 61,A 171.8226,B 24.8426,C -2.8944,E1 24.8399,E2 -448.6965} C_DIS
LIN {X -36.1177,Y 2.5391,Z 61,A 168.1474,B 24.8419,C -2.9007,E1 24.8404,E2 -445.0143} C_DIS
LIN {X -35.9326,Y 4.4491,Z 61,A 165.3673,B 24.8406,C -2.9124,E1 24.8412,E2 -442.2457} C_DIS
LIN {X -35.7051,Y 6.0071,Z 61,A 163.0028,B 24.8396,C -2.9213,E1 24.8422,E2 -439.8883} C_DIS
LIN {X -35.0978,Y 8.8914,Z 61,A 157.3755,B 24.839,C -2.9273,E1 24.8458,E2 -434.2424} C_DIS
LIN {X -34.3331,Y 11.4973,Z 61,A 153.7901,B 24.8368,C -2.9466,E1 24.8487,E2 -430.6826} C_DIS
LIN {X -33.5852,Y 13.5275,Z 61,A 150.1097,B 24.8359,C -2.9546,E1 24.8524,E2 -427.0006} C_DIS
LIN {X -32.5271,Y 15.9041,Z 61,A 145.705,B 24.8349,C -2.964,E1 24.8576,E2 -422.5945} C_DIS
LIN {X -31.5108,Y 17.834,Z 61,A 142.8553,B 24.8332,C -2.9792,E1 24.8614,E2 -419.7662} C_DIS
LIN {X -30.3958,Y 19.6737,Z 61,A 138.8294,B 24.8328,C -2.983,E1 24.8674,E2 -415.7287} C_DIS
LIN {X -29.1278,Y 21.5066,Z 61,A 135.8522,B 24.8311,C -2.9974,E1 24.8722,E2 -412.7714} C_DIS
LIN {X -27.484,Y 23.5708,Z 61,A 130.68,B 24.831,C -2.9987,E1 24.8814,E2 -407.5786} C_DIS
LIN {X -25.5724,Y 25.6318,Z 61,A 126.1816,B 24.8298,C -3.0088,E1 24.8902,E2 -403.085} C_DIS
LIN {X -22.5638,Y 28.3165,Z 61,A 120.4261,B 24.8276,C -3.0287,E1 24.9024,E2 -397.3548} C_DIS
LIN {X -20.2743,Y 29.9982,Z 61,A 115.5334,B 24.827,C -3.0336,E1 24.9136,E2 -392.457} C_DIS
LIN {X -17.931,Y 31.4553,Z 61,A 111.1502,B 24.8262,C -3.0411,E1 24.9241,E2 -388.0785} C_DIS
LIN {X -15.0709,Y 32.9217,Z 61,A 106.539,B 24.8247,C -3.0538,E1 24.9356,E2 -383.4856} C_DIS
LIN {X -13.1528,Y 33.7336,Z 61,A 103.2175,B 24.8242,C -3.0581,E1 24.9442,E2 -380.1668} C_DIS
LIN {X -11.145,Y 34.449,Z 61,A 99.841,B 24.8237,C -3.062,E1 24.9531,E2 -376.7934} C_DIS
LIN {X -9.0102,Y 35.0677,Z 61,A 96.7128,B 24.8228,C -3.0699,E1 24.9615,E2 -373.6789} C_DIS
LIN {X -7.7742,Y 35.3625,Z 61,A 94.2498,B 24.8232,C -3.0666,E1 24.9682,E2 -371.2051} C_DIS
LIN {X -6.0177,Y 35.7034,Z 61,A 91.3593,B 24.823,C -3.0681,E1 24.9762,E2 -368.3151} C_DIS
LIN {X -3.888,Y 35.9978,Z 61,A 88.0413,B 24.8227,C -3.071,E1 24.9854,E2 -365.0017} C_DIS
LIN {X -1.6414,Y 36.1697,Z 61,A 84.3966,B 24.8227,C -3.0714,E1 24.9955,E2 -361.3569} C_DIS
LIN {X 0.7143,Y 36.1999,Z 61,A 80.6966,B 24.8225,C -3.0725,E1 25.0058,E2 -357.6595} C_DIS
LIN {X 2.7077,Y 36.106,Z 61,A 77.1571,B 24.8231,C -3.0679,E1 25.0157,E2 -354.1107} C_DIS
LIN {X 4.8526,Y 35.8806,Z 61,A 73.5299,B 24.8234,C -3.0646,E1 25.0258,E2 -350.4786} C_DIS
LIN {X 8.5495,Y 35.1831,Z 61,A 68.4896,B 24.8224,C -3.0732,E1 25.0395,E2 -345.465} C_DIS
LIN {X 10.8859,Y 34.532,Z 61,A 63.9722,B 24.8237,C -3.062,E1 25.0516,E2 -340.9288} C_DIS
LIN {X 13.0798,Y 33.7622,Z 61,A 60.9424,B 24.8232,C -3.067,E1 25.0595,E2 -337.9172} C_DIS
LIN {X 14.8419,Y 33.0252,Z 61,A 57.6233,B 24.824,C -3.0599,E1 25.068,E2 -334.5894} C_DIS
LIN {X 16.4497,Y 32.2545,Z 61,A 55.2264,B 24.8237,C -3.0621,E1 25.074,E2 -332.204} C_DIS
LIN {X 17.7885,Y 31.5362,Z 61,A 52.6507,B 24.8244,C -3.0566,E1 25.0803,E2 -329.6228} C_DIS
LIN {X 19.1197,Y 30.7471,Z 61,A 49.8902,B 24.8253,C -3.0488,E1 25.0869,E2 -326.8526} C_DIS
LIN {X 21.2938,Y 29.2836,Z 61,A 45.98,B 24.8257,C -3.0453,E1 25.0959,E2 -322.9474} C_DIS
LIN {X 22.6108,Y 28.2793,Z 61,A 43.5831,B 24.8258,C -3.0438,E1 25.1011,E2 -320.5556} C_DIS
LIN {X 23.9662,Y 27.1401,Z 61,A 40.4874,B 24.8269,C -3.0344,E1 25.1077,E2 -317.4499} C_DIS
LIN {X 25.5001,Y 25.7039,Z 61,A 37.1983,B 24.8276,C -3.0282,E1 25.1143,E2 -314.1597} C_DIS
LIN {X 26.7306,Y 24.4218,Z 61,A 34.6442,B 24.8279,C -3.0258,E1 25.1192,E2 -311.611} C_DIS
LIN {X 27.6251,Y 23.4053,Z 61,A 32.603,B 24.8283,C -3.0224,E1 25.1229,E2 -309.5711} C_DIS
LIN {X 28.4725,Y 22.3667,Z 61,A 30.0458,B 24.8296,C -3.0113,E1 25.1274,E2 -306.9994} C_DIS
LIN {X 29.448,Y 21.0656,Z 61,A 27.3457,B 24.8305,C -3.0032,E1 25.1318,E2 -304.2933} C_DIS
LIN {X 30.993,Y 18.7186,Z 61,A 23.3656,B 24.831,C -2.9987,E1 25.1378,E2 -300.3227} C_DIS
LIN {X 32.2012,Y 16.5539,Z 61,A 18.7282,B 24.8333,C -2.9779,E1 25.1439,E2 -295.6602} C_DIS
LIN {X 33.396,Y 13.9875,Z 61,A 14.4642,B 24.8344,C -2.9686,E1 25.1487,E2 -291.3975} C_DIS
LIN {X 34.4613,Y 11.1069,Z 61,A 10.0491,B 24.8352,C -2.9612,E1 25.1528,E2 -286.9897} C_DIS
LIN {X 35.1248,Y 8.785,Z 61,A 5.6155,B 24.8375,C -2.9407,E1 25.1559,E2 -282.533} C_DIS
LIN {X 35.6556,Y 6.2953,Z 61,A 1.856,B 24.8384,C -2.9325,E1 25.1579,E2 -278.7761} C_DIS
LIN {X 36.0361,Y 3.5181,Z 61,A -2.0016,B 24.8389,C -2.9275,E1 25.1592,E2 -274.9296} C_DIS
LIN {X 36.17,Y 1.6376,Z 61,A -5.0762,B 24.8401,C -2.9169,E1 25.1597,E2 -271.848} C_DIS
LIN {X 36.202,Y -0.5464,Z 61,A -9.0011,B 24.8421,C -2.899,E1 25.1597,E2 -267.9041} C_DIS
LIN {X 35.9384,Y -4.3989,Z 61,A -15.3223,B 24.8445,C -2.8767,E1 25.158,E2 -261.5676} C_DIS
LIN {X 35.4504,Y -7.3631,Z 61,A -19.4734,B 24.8451,C -2.8709,E1 25.1559,E2 -257.4272} C_DIS
LIN {X 34.9547,Y -9.4398,Z 61,A -22.6351,B 24.8459,C -2.8638,E1 25.1537,E2 -254.2668} C_DIS
LIN {X 34.2554,Y -11.7272,Z 61,A -26.9335,B 24.848,C -2.8445,E1 25.15,E2 -249.9472} C_DIS
LIN {X 33.2845,Y -14.2523,Z 61,A -30.5364,B 24.8483,C -2.8419,E1 25.1463,E2 -246.358} C_DIS
LIN {X 32.7394,Y -15.4616,Z 61,A -32.9323,B 24.8494,C -2.8313,E1 25.1434,E2 -243.95} C_DIS
LIN {X 31.6296,Y -17.6213,Z 61,A -36.6667,B 24.8504,C -2.8219,E1 25.1385,E2 -240.213} C_DIS
LIN {X 30.3546,Y -19.7378,Z 61,A -40.7924,B 24.8519,C -2.8079,E1 25.1324,E2 -236.0749} C_DIS
LIN {X 29.2112,Y -21.3928,Z 61,A -43.8203,B 24.8525,C -2.8017,E1 25.1275,E2 -233.047} C_DIS
LIN {X 28.2027,Y -22.706,Z 61,A -46.3752,B 24.8532,C -2.7958,E1 25.123,E2 -230.4902} C_DIS
LIN {X 26.6909,Y -24.465,Z 61,A -49.8109,B 24.8538,C -2.7901,E1 25.1167,E2 -227.0564} C_DIS
LIN {X 25.4249,Y -25.7782,Z 61,A -52.6803,B 24.8545,C -2.7835,E1 25.111,E2 -224.1835} C_DIS
LIN {X 24.1221,Y -27.0013,Z 61,A -55.5885,B 24.8553,C -2.7759,E1 25.105,E2 -221.269} C_DIS
LIN {X 22.8203,Y -28.1101,Z 61,A -58.4042,B 24.856,C -2.7684,E1 25.099,E2 -218.4465} C_DIS
LIN {X 20.9589,Y -29.5241,Z 61,A -61.8146,B 24.8564,C -2.765,E1 25.0913,E2 -215.04} C_DIS
LIN {X 19.7522,Y -30.3448,Z 61,A -63.9423,B 24.8566,C -2.7631,E1 25.0864,E2 -212.9149} C_DIS
LIN {X 18.0011,Y -31.415,Z 61,A -67.9179,B 24.8583,C -2.7472,E1 25.0768,E2 -208.9137} C_DIS
LIN {X 16.0379,Y -32.4612,Z 61,A -70.8126,B 24.858,C -2.75,E1 25.0696,E2 -206.0338} C_DIS
LIN {X 14.7875,Y -33.0496,Z 61,A -73.3677,B 24.8588,C -2.7417,E1 25.0631,E2 -203.4654} C_DIS
LIN {X 12.4395,Y -34.003,Z 61,A -77.0133,B 24.8588,C -2.7412,E1 25.0536,E2 -199.8266} C_DIS
LIN {X 10.91,Y -34.5245,Z 61,A -79.5851,B 24.8592,C -2.7379,E1 25.0468,E2 -197.2519} C_DIS
LIN {X 9.3064,Y -34.9907,Z 61,A -82.2737,B 24.8596,C -2.7345,E1 25.0396,E2 -194.5596} C_DIS
LIN {X 7.3075,Y -35.4618,Z 61,A -85.7859,B 24.8602,C -2.7282,E1 25.0299,E2 -191.0371} C_DIS
LIN {X 5.3883,Y -35.8038,Z 61,A -88.8817,B 24.8605,C -2.7258,E1 25.0214,E2 -187.9387} C_DIS
LIN {X 2.7724,Y -36.1008,Z 61,A -93.0683,B 24.8607,C -2.7234,E1 25.0098,E2 -183.7489} C_DIS
LIN {X 0.6403,Y -36.2013,Z 61,A -96.3081,B 24.8607,C -2.724,E1 25.0007,E2 -180.5113} C_DIS
LIN {X 0.6403,Y -36.2013,Z 61,A -96.3081,B 24.8607,C -2.724,E1 25.0007,E2 -180.5113} C_DIS
Enddeposition()
LIN {X 0.2057,Y -35.218,Z 61,A -96.0201,B 24.8577,C -2.7529,E1 25.0017,E2 -180.8681} C_DIS
Startdeposition()
$VEL.CP = VEL_PRINT
LIN {X 1.6954,Y -35.1816,Z 61,A -93.056,B 24.8569,C -2.7603,E1 25.01,E2 -183.8491} C_DIS
LIN {X 4.2484,Y -34.9651,Z 61,A -88.7983,B 24.8565,C -2.7637,E1 25.0219,E2 -188.1121} C_DIS
LIN {X 6.451,Y -34.6265,Z 61,A -84.6999,B 24.8556,C -2.7725,E1 25.0332,E2 -192.2271} C_DIS
LIN {X 8.284,Y -34.2339,Z 61,A -81.8089,B 24.8556,C -2.7733,E1 25.0411,E2 -195.1159} C_DIS
LIN {X 10.9263,Y -33.4844,Z 61,A -77.9035,B 24.8558,C -2.7709,E1 25.0515,E2 -199.0087} C_DIS
LIN {X 12.265,Y -33.0177,Z 61,A -74.6841,B 24.8542,C -2.7862,E1 25.06,E2 -202.2576} C_DIS
LIN {X 16.0125,Y -31.3717,Z 61,A -68.9699,B 24.8545,C -2.7834,E1 25.0744,E2 -207.9506} C_DIS
LIN {X 17.082,Y -30.8016,Z 61,A -66.5114,B 24.8534,C -2.7935,E1 25.0804,E2 -210.4259} C_DIS
LIN {X 19.5147,Y -29.3216,Z 61,A -62.275,B 24.8531,C -2.7965,E1 25.0904,E2 -214.656} C_DIS
LIN {X 20.8927,Y -28.3563,Z 61,A -59.7073,B 24.8528,C -2.7997,E1 25.0963,E2 -217.2221} C_DIS
LIN {X 22.1659,Y -27.3725,Z 61,A -56.8979,B 24.8519,C -2.8079,E1 25.1024,E2 -220.0407} C_DIS
LIN {X 23.5051,Y -26.2315,Z 61,A -54.1279,B 24.8514,C -2.813,E1 25.1083,E2 -222.8118} C_DIS
LIN {X 24.7479,Y -25.0624,Z 61,A -51.3303,B 24.8506,C -2.8198,E1 25.1139,E2 -225.6139} C_DIS
LIN {X 25.8993,Y -23.8708,Z 61,A -48.7235,B 24.8501,C -2.8251,E1 25.1189,E2 -228.2217} C_DIS
LIN {X 26.936,Y -22.6948,Z 61,A -46.1293,B 24.8493,C -2.8321,E1 25.1236,E2 -230.8209} C_DIS
LIN {X 28.2287,Y -21.0638,Z 61,A -42.0177,B 24.8472,C -2.8517,E1 25.1306,E2 -234.9594} C_DIS
LIN {X 30.4485,Y -17.706,Z 61,A -35.2602,B 24.8449,C -2.873,E1 25.1406,E2 -241.733} C_DIS
LIN {X 32.296,Y -14.0553,Z 61,A -29.4994,B 24.8443,C -2.8789,E1 25.1475,E2 -247.4769} C_DIS
LIN {X 33.059,Y -12.1527,Z 61,A -26.1727,B 24.8432,C -2.8888,E1 25.1508,E2 -250.8085} C_DIS
LIN {X 33.5737,Y -10.6503,Z 61,A -23.9744,B 24.843,C -2.8908,E1 25.1527,E2 -252.9991} C_DIS
LIN {X 34.089,Y -8.8619,Z 61,A -20.4284,B 24.8411,C -2.908,E1 25.1554,E2 -256.5654} C_DIS
LIN {X 34.5468,Y -6.8662,Z 61,A -17.4938,B 24.8406,C -2.9123,E1 25.1571,E2 -259.4932} C_DIS
LIN {X 34.9033,Y -4.7289,Z 61,A -13.4368,B 24.8385,C -2.9314,E1 25.1588,E2 -263.5715} C_DIS
LIN {X 35.1431,Y -2.3548,Z 61,A -9.9359,B 24.8378,C -2.9378,E1 25.1596,E2 -267.0668} C_DIS
LIN {X 35.2202,Y -0.3761,Z 61,A -6.8692,B 24.837,C -2.9456,E1 25.1598,E2 -270.1336} C_DIS
LIN {X 35.2029,Y 1.1588,Z 61,A -4.5371,B 24.8364,C -2.9509,E1 25.1596,E2 -272.4644} C_DIS
LIN {X 35.125,Y 2.6164,Z 61,A -2.1422,B 24.8355,C -2.9586,E1 25.1592,E2 -274.8632} C_DIS
LIN {X 34.9335,Y 4.4986,Z 61,A 1.3792,B 24.8337,C -2.9748,E1 25.158,E2 -278.4021} C_DIS
LIN {X 34.6547,Y 6.2956,Z 61,A 4.3951,B 24.8326,C -2.9846,E1 25.1566,E2 -281.4238} C_DIS
LIN {X 34.0739,Y 8.9167,Z 61,A 8.0517,B 24.8323,C -2.9871,E1 25.1542,E2 -285.0649} C_DIS
LIN {X 33.6093,Y 10.5363,Z 61,A 11.832,B 24.8296,C -3.0106,E1 25.1511,E2 -288.8796} C_DIS
LIN {X 32.3395,Y 13.9555,Z 61,A 16.7497,B 24.8294,C -3.0123,E1 25.1461,E2 -293.774} C_DIS
LIN {X 31.7723,Y 15.2023,Z 61,A 19.3386,B 24.8281,C -3.0238,E1 25.143,E2 -296.376} C_DIS
LIN {X 30.6807,Y 17.3001,Z 61,A 22.7643,B 24.8277,C -3.0278,E1 25.1385,E2 -299.7934} C_DIS
LIN {X 30.0385,Y 18.3925,Z 61,A 25.2342,B 24.8264,C -3.039,E1 25.1349,E2 -302.2772} C_DIS
LIN {X 28.7375,Y 20.3655,Z 61,A 28.9804,B 24.8255,C -3.0471,E1 25.129,E2 -306.0241} C_DIS
LIN {X 27.5306,Y 21.9699,Z 61,A 32.1639,B 24.8247,C -3.0536,E1 25.1236,E2 -309.2079} C_DIS
LIN {X 26.5282,Y 23.1698,Z 61,A 34.4362,B 24.8245,C -3.0555,E1 25.1194,E2 -311.4744} C_DIS
LIN {X 25.0068,Y 24.8037,Z 61,A 38.5381,B 24.8228,C -3.0698,E1 25.1115,E2 -315.5924} C_DIS
LIN {X 23.0314,Y 26.648,Z 61,A 43.1905,B 24.8214,C -3.0818,E1 25.1018,E2 -320.2549} C_DIS
LIN {X 21.0695,Y 28.2254,Z 61,A 47.3128,B 24.8206,C -3.0893,E1 25.0926,E2 -324.3799} C_DIS
LIN {X 18.3975,Y 30.0355,Z 61,A 51.7076,B 24.821,C -3.0859,E1 25.0824,E2 -328.7521} C_DIS
LIN {X 17.3023,Y 30.6796,Z 61,A 53.915,B 24.8204,C -3.0906,E1 25.0771,E2 -330.9641} C_DIS
LIN {X 15.797,Y 31.481,Z 61,A 56.6021,B 24.8201,C -3.093,E1 25.0704,E2 -333.6493} C_DIS
LIN {X 14.5433,Y 32.0793,Z 61,A 58.7541,B 24.8201,C -3.0942,E1 25.065,E2 -335.7987} C_DIS
LIN {X 12.78,Y 32.8217,Z 61,A 62.3809,B 24.8189,C -3.1039,E1 25.0555,E2 -339.4403} C_DIS
LIN {X 10.5703,Y 33.5987,Z 61,A 66.1067,B 24.8186,C -3.1059,E1 25.0457,E2 -343.1636} C_DIS
LIN {X 8.5861,Y 34.1598,Z 61,A 69.2526,B 24.8187,C -3.1053,E1 25.0372,E2 -346.3033} C_DIS
LIN {X 6.3971,Y 34.6365,Z 61,A 73.2762,B 24.818,C -3.1115,E1 25.0262,E2 -350.3368} C_DIS
LIN {X 4.2475,Y 34.9651,Z 61,A 76.4214,B 24.8184,C -3.1076,E1 25.0175,E2 -353.47} C_DIS
LIN {X 2.5067,Y 35.1328,Z 61,A 79.2319,B 24.8184,C -3.1074,E1 25.0097,E2 -356.2785} C_DIS
LIN {X 0.5146,Y 35.2184,Z 61,A 82.8596,B 24.818,C -3.1115,E1 24.9995,E2 -359.9153} C_DIS
LIN {X -1.5073,Y 35.1896,Z 61,A 86.2552,B 24.818,C -3.1118,E1 24.9901,E2 -363.3121} C_DIS
LIN {X -4.0942,Y 34.9831,Z 61,A 90.3412,B 24.8184,C -3.1081,E1 24.9787,E2 -367.3917} C_DIS
LIN {X -6.8329,Y 34.5532,Z 61,A 94.2149,B 24.8196,C -3.0978,E1 24.9681,E2 -371.2445} C_DIS
LIN {X -9.2303,Y 33.991,Z 61,A 99.2981,B 24.8186,C -3.1058,E1 24.9543,E2 -376.354} C_DIS
LIN {X -11.6619,Y 33.2353,Z 61,A 102.6296,B 24.8202,C -3.0923,E1 24.9455,E2 -379.6594} C_DIS
LIN {X -13.6873,Y 32.4536,Z 61,A 106.6075,B 24.8202,C -3.0922,E1 24.9352,E2 -383.6458} C_DIS
LIN {X -16.0251,Y 31.3652,Z 61,A 110.8299,B 24.821,C -3.086,E1 24.9246,E2 -387.8644} C_DIS
LIN {X -17.9319,Y 30.3155,Z 61,A 114.0195,B 24.8221,C -3.0763,E1 24.9169,E2 -391.0404} C_DIS
LIN {X -19.5087,Y 29.326,Z 61,A 117.1368,B 24.8226,C -3.0716,E1 24.9096,E2 -394.1564} C_DIS
LIN {X -21.3677,Y 28.0006,Z 61,A 121.1383,B 24.8232,C -3.067,E1 24.9006,E2 -398.161} C_DIS
LIN {X -23.3899,Y 26.3347,Z 61,A 125.4765,B 24.8242,C -3.0584,E1 24.8914,E2 -402.4957} C_DIS
LIN {X -25.1707,Y 24.6382,Z 61,A 129.3028,B 24.8254,C -3.0474,E1 24.8838,E2 -406.3117} C_DIS
LIN {X -26.7977,Y 22.8575,Z 61,A 133.3541,B 24.8264,C -3.0389,E1 24.8764,E2 -410.3609} C_DIS
LIN {X -28.4696,Y 20.7381,Z 61,A 138.0077,B 24.8274,C -3.0299,E1 24.8685,E2 -415.0152} C_DIS
LIN {X -29.7488,Y 18.8581,Z 61,A 141.1375,B 24.8292,C -3.0146,E1 24.8638,E2 -418.1241} C_DIS
LIN {X -30.6608,Y 17.336,Z 61,A 144.1779,B 24.8299,C -3.0079,E1 24.8595,E2 -421.1643} C_DIS
LIN {X -31.6569,Y 15.4418,Z 61,A 147.816,B 24.8309,C -2.9993,E1 24.8549,E2 -424.8013} C_DIS
LIN {X -32.7137,Y 13.0537,Z 61,A 152.4916,B 24.8319,C -2.9906,E1 24.8499,E2 -429.482} C_DIS
LIN {X -33.6203,Y 10.5005,Z 61,A 156.6817,B 24.8336,C -2.9753,E1 24.8462,E2 -433.6594} C_DIS
LIN {X -34.3166,Y 7.9337,Z 61,A 160.8334,B 24.8353,C -2.9604,E1 24.8434,E2 -437.7998} C_DIS
LIN {X -34.7308,Y 5.8616,Z 61,A 164.249,B 24.8365,C -2.9495,E1 24.8416,E2 -441.2096} C_DIS
LIN {X -35.0042,Y 3.9142,Z 61,A 167.3477,B 24.8377,C -2.9387,E1 24.8406,E2 -444.3008} C_DIS
LIN {X -35.1571,Y 2.141,Z 61,A 170.4917,B 24.8385,C -2.9318,E1 24.8399,E2 -447.4471} C_DIS
LIN {X -35.2204,Y 0.2841,Z 61,A 173.1186,B 24.8399,C -2.9189,E1 24.8398,E2 -450.059} C_DIS
LIN {X -35.2043,Y -1.1125,Z 61,A 175.4822,B 24.8406,C -2.9126,E1 24.8399,E2 -452.4218} C_DIS
LIN {X -35.1118,Y -2.783,Z 61,A 178.4332,B 24.8413,C -2.9062,E1 24.8405,E2 -455.3751} C_DIS
LIN {X -34.904,Y -4.7257,Z 61,A -178.3633,B 24.8423,C -2.8966,E1 24.8416,E2 -458.5749} C_DIS
LIN {X -34.5847,Y -6.6695,Z 61,A -175.1439,B 24.8434,C -2.887,E1 24.8431,E2 -461.7904} C_DIS
LIN {X -34.2486,Y -8.224,Z 61,A -172.7583,B 24.8444,C -2.8775,E1 24.8446,E2 -464.1672} C_DIS
LIN {X -33.7239,Y -10.1632,Z 61,A -169.2684,B 24.8453,C -2.8698,E1 24.8473,E2 -467.659} C_DIS
LIN {X -32.8745,Y -12.644,Z 61,A -164.3039,B 24.8459,C -2.864,E1 24.852,E2 -472.6375} C_DIS
LIN {X -31.7265,Y -15.2975,Z 61,A -160.2396,B 24.8479,C -2.8451,E1 24.8567,E2 -476.679} C_DIS
LIN {X -31.0113,Y -16.7001,Z 61,A -157.8184,B 24.8488,C -2.837,E1 24.8599,E2 -479.0937} C_DIS
LIN {X -30.3034,Y -17.9524,Z 61,A -155.4483,B 24.8494,C -2.8312,E1 24.8632,E2 -481.4623} C_DIS
LIN {X -29.4945,Y -19.2531,Z 61,A -152.9975,B 24.8501,C -2.8245,E1 24.8668,E2 -483.9096} C_DIS
LIN {X -28.7103,Y -20.4036,Z 61,A -150.7584,B 24.8507,C -2.8188,E1 24.8704,E2 -486.1459} C_DIS
LIN {X -27.9944,Y -21.3756,Z 61,A -147.9497,B 24.8504,C -2.8223,E1 24.8752,E2 -488.9764} C_DIS
LIN {X -26.0438,Y -23.7133,Z 61,A -143.1554,B 24.8517,C -2.8098,E1 24.884,E2 -493.7624} C_DIS
LIN {X -23.8091,Y -25.9559,Z 61,A -138.5114,B 24.8533,C -2.7943,E1 24.8933,E2 -498.3888} C_DIS
LIN {X -21.9867,Y -27.5171,Z 61,A -134.0057,B 24.8534,C -2.7933,E1 24.903,E2 -502.9093} C_DIS
LIN {X -19.9373,Y -29.0366,Z 61,A -130.1886,B 24.8545,C -2.7831,E1 24.9116,E2 -506.7152} C_DIS
LIN {X -18.0891,Y -30.2225,Z 61,A -126.5487,B 24.855,C -2.7786,E1 24.9203,E2 -510.3558} C_DIS
LIN {X -15.7309,Y -31.514,Z 61,A -121.9667,B 24.8553,C -2.7754,E1 24.9316,E2 -514.9427} C_DIS
LIN {X -13.5101,Y -32.5283,Z 61,A -118.1824,B 24.856,C -2.7692,E1 24.9413,E2 -518.7212} C_DIS
LIN {X -11.6506,Y -33.2392,Z 61,A -115.1892,B 24.8565,C -2.7636,E1 24.9491,E2 -521.7072} C_DIS
LIN {X -9.4541,Y -33.9297,Z 61,A -110.8675,B 24.8561,C -2.7677,E1 24.9607,E2 -526.0458} C_DIS
LIN {X -6.8859,Y -34.5421,Z 61,A -107.0103,B 24.8569,C -2.7607,E1 24.9712,E2 -529.8911} C_DIS
LIN {X -4.798,Y -34.8939,Z 61,A -104.0348,B 24.8575,C -2.7543,E1 24.9794,E2 -532.854} C_DIS
LIN {X -2.4567,Y -35.1362,Z 61,A -99.6221,B 24.8568,C -2.761,E1 24.9917,E2 -537.285} C_DIS
LIN {X -0.1861,Y -35.2214,Z 61,A -96.0374,B 24.8568,C -2.7602,E1 25.0017,E2 -540.8681} C_DIS
LIN {X -0.1861,Y -35.2214,Z 61,A -96.0374,B 24.8568,C -2.7602,E1 25.0017,E2 -540.8681} C_DIS
Enddeposition()
LIN {X 0.2015,Y -34.2309,Z 61,A -96.3126,B 24.8562,C -2.7665,E1 25.001,E2 -540.6078} C_DIS
Startdeposition()
$VEL.CP = VEL_PRINT
LIN {X -1.507,Y -34.2037,Z 61,A -99.6736,B 24.8569,C -2.7601,E1 24.9916,E2 -537.2314} C_DIS
LIN {X -3.4962,Y -34.058,Z 61,A -103.3134,B 24.8572,C -2.7568,E1 24.9814,E2 -533.5821} C_DIS
LIN {X -5.3185,Y -33.8214,Z 61,A -106.0946,B 24.8568,C -2.7608,E1 24.9738,E2 -530.808} C_DIS
LIN {X -7.1268,Y -33.4874,Z 61,A -109.4707,B 24.8571,C -2.7587,E1 24.9645,E2 -527.423} C_DIS
LIN {X -9.1367,Y -32.9958,Z 61,A -112.8602,B 24.8568,C -2.7614,E1 24.9553,E2 -524.0352} C_DIS
LIN {X -11.346,Y -32.3022,Z 61,A -117.0841,B 24.8568,C -2.7608,E1 24.9441,E2 -519.8017} C_DIS
LIN {X -13.7171,Y -31.3689,Z 61,A -121.3774,B 24.8564,C -2.7647,E1 24.9331,E2 -515.5081} C_DIS
LIN {X -16.3822,Y -30.063,Z 61,A -126.0973,B 24.8555,C -2.7733,E1 24.9213,E2 -510.7959} C_DIS
LIN {X -18.4431,Y -28.8448,Z 61,A -130.1847,B 24.855,C -2.7783,E1 24.9116,E2 -506.7077} C_DIS
LIN {X -20.0761,Y -27.7334,Z 61,A -133.4942,B 24.8545,C -2.7836,E1 24.9041,E2 -503.3995} C_DIS
LIN {X -21.9142,Y -26.3045,Z 61,A -136.8664,B 24.8532,C -2.7955,E1 24.8967,E2 -500.0433} C_DIS
LIN {X -22.8386,Y -25.5061,Z 61,A -139.298,B 24.8532,C -2.7958,E1 24.8916,E2 -497.6026} C_DIS
LIN {X -24.5228,Y -23.8916,Z 61,A -143.3782,B 24.8525,C -2.8021,E1 24.8835,E2 -493.5203} C_DIS
LIN {X -26.1003,Y -22.1572,Z 61,A -147.3894,B 24.8517,C -2.81,E1 24.8761,E2 -489.5099} C_DIS
LIN {X -27.2423,Y -20.7379,Z 61,A -149.9502,B 24.8505,C -2.8214,E1 24.8718,E2 -486.9643} C_DIS
LIN {X -28.4922,Y -18.9838,Z 61,A -154.0573,B 24.85,C -2.8258,E1 24.8652,E2 -482.8475} C_DIS
LIN {X -29.58,Y -17.2396,Z 61,A -157.3299,B 24.8489,C -2.8361,E1 24.8605,E2 -479.5826} C_DIS
LIN {X -30.5726,Y -15.4109,Z 61,A -160.9231,B 24.848,C -2.8444,E1 24.8559,E2 -475.9902} C_DIS
LIN {X -31.2748,Y -13.9304,Z 61,A -164.2325,B 24.8477,C -2.8472,E1 24.8521,E2 -472.6693} C_DIS
LIN {X -32.6184,Y -10.4032,Z 61,A -170.5146,B 24.8457,C -2.8657,E1 24.8462,E2 -466.3957} C_DIS
LIN {X -33.4079,Y -7.4911,Z 61,A -174.868,B 24.8435,C -2.8864,E1 24.8433,E2 -462.0666} C_DIS
LIN {X -33.7255,Y -5.8933,Z 61,A -177.498,B 24.8425,C -2.8955,E1 24.8419,E2 -459.4428} C_DIS
LIN {X -33.9285,Y -4.5887,Z 61,A 179.7519,B 24.8422,C -2.8978,E1 24.8409,E2 -456.6818} C_DIS
LIN {X -34.1856,Y -1.8728,Z 61,A 175.8149,B 24.8401,C -2.9171,E1 24.84,E2 -452.7673} C_DIS
LIN {X -34.2357,Y 0.0186,Z 61,A 172.1323,B 24.8395,C -2.9228,E1 24.8398,E2 -449.0761} C_DIS
LIN {X -34.1708,Y 2.126,Z 61,A 168.5861,B 24.8383,C -2.9337,E1 24.8403,E2 -445.5346} C_DIS
LIN {X -33.9924,Y 4.0854,Z 61,A 165.3544,B 24.8371,C -2.9445,E1 24.8412,E2 -442.3094} C_DIS
LIN {X -33.6892,Y 6.0994,Z 61,A 161.9212,B 24.8359,C -2.9549,E1 24.8428,E2 -438.8807} C_DIS
LIN {X -33.261,Y 8.116,Z 61,A 158.2583,B 24.8349,C -2.9638,E1 24.845,E2 -435.2177} C_DIS
LIN {X -32.8221,Y 9.7403,Z 61,A 155.5953,B 24.8338,C -2.9737,E1 24.8471,E2 -432.5629} C_DIS
LIN {X -31.8427,Y 12.5781,Z 61,A 149.8836,B 24.8327,C -2.9832,E1 24.8526,E2 -426.8417} C_DIS
LIN {X -30.7881,Y 14.9762,Z 61,A 146.2266,B 24.8306,C -3.0019,E1 24.8569,E2 -423.2096} C_DIS
LIN {X -29.8286,Y 16.8056,Z 61,A 142.3252,B 24.8299,C -3.008,E1 24.8621,E2 -419.3023} C_DIS
LIN {X -27.7765,Y 20.0151,Z 61,A 135.3277,B 24.8286,C -3.0201,E1 24.873,E2 -412.2987} C_DIS
LIN {X -26.1192,Y 22.1351,Z 61,A 132.0005,B 24.8261,C -3.0416,E1 24.8788,E2 -409.0075} C_DIS
LIN {X -24.4848,Y 23.931,Z 61,A 126.9183,B 24.826,C -3.0425,E1 24.8886,E2 -403.9054} C_DIS
LIN {X -22.6923,Y 25.6371,Z 61,A 123.6573,B 24.824,C -3.0596,E1 24.8952,E2 -400.6721} C_DIS
LIN {X -20.636,Y 27.319,Z 61,A 118.0234,B 24.8242,C -3.0582,E1 24.9077,E2 -395.0141} C_DIS
LIN {X -18.6975,Y 28.681,Z 61,A 114.5436,B 24.8228,C -3.0701,E1 24.9157,E2 -391.5512} C_DIS
LIN {X -16.4713,Y 30.0145,Z 61,A 110.5979,B 24.8215,C -3.0813,E1 24.9252,E2 -387.6207} C_DIS
LIN {X -14.7151,Y 30.9135,Z 61,A 106.7837,B 24.8215,C -3.0815,E1 24.9348,E2 -383.797} C_DIS
LIN {X -11.5894,Y 32.216,Z 61,A 101.7436,B 24.8199,C -3.0952,E1 24.9478,E2 -378.7786} C_DIS
LIN {X -9.6972,Y 32.8349,Z 61,A 98.1702,B 24.8197,C -3.0965,E1 24.9574,E2 -375.202} C_DIS
LIN {X -7.9763,Y 33.2951,Z 61,A 95.4739,B 24.8191,C -3.1022,E1 24.9646,E2 -372.5156} C_DIS
LIN {X -6.6514,Y 33.5851,Z 61,A 93.2919,B 24.8187,C -3.105,E1 24.9706,E2 -370.3376} C_DIS
LIN {X -5.1577,Y 33.8462,Z 61,A 90.5726,B 24.8187,C -3.1049,E1 24.9781,E2 -367.6154} C_DIS
LIN {X -3.453,Y 34.0625,Z 61,A 87.6943,B 24.8186,C -3.1064,E1 24.9861,E2 -364.7389} C_DIS
LIN {X -1.9859,Y 34.1794,Z 61,A 85.4424,B 24.8182,C -3.1097,E1 24.9923,E2 -362.494} C_DIS
LIN {X -0.6478,Y 34.2308,Z 61,A 83.1323,B 24.8182,C -3.1096,E1 24.9988,E2 -360.1833} C_DIS
LIN {X 0.7561,Y 34.2288,Z 61,A 80.7387,B 24.8182,C -3.1094,E1 25.0055,E2 -357.7897} C_DIS
LIN {X 2.4669,Y 34.1476,Z 61,A 77.3173,B 24.8189,C -3.1032,E1 25.015,E2 -354.3549} C_DIS
LIN {X 5.2514,Y 33.8317,Z 61,A 73.1133,B 24.8184,C -3.1078,E1 25.0266,E2 -350.1652} C_DIS
LIN {X 6.8786,Y 33.5388,Z 61,A 69.8815,B 24.8192,C -3.1012,E1 25.0355,E2 -346.9216} C_DIS
LIN {X 9.6792,Y 32.8402,Z 61,A 65.7195,B 24.8186,C -3.1062,E1 25.0467,E2 -342.7779} C_DIS
LIN {X 10.8291,Y 32.4792,Z 61,A 62.7488,B 24.8201,C -3.0931,E1 25.0547,E2 -339.7819} C_DIS
LIN {X 14.2394,Y 31.1358,Z 61,A 57.7607,B 24.8192,C -3.101,E1 25.0674,E2 -334.8239} C_DIS
LIN {X 15.74,Y 30.4043,Z 61,A 54.2905,B 24.8206,C -3.0891,E1 25.0762,E2 -331.335} C_DIS
LIN {X 17.674,Y 29.3225,Z 61,A 50.299,B 24.8216,C -3.0803,E1 25.0858,E2 -327.3348} C_DIS
LIN {X 20.3815,Y 27.5096,Z 61,A 45.6421,B 24.8215,C -3.0817,E1 25.0964,E2 -322.6971} C_DIS
LIN {X 22.2682,Y 26.0045,Z 61,A 40.9688,B 24.8233,C -3.0661,E1 25.1066,E2 -318.0045} C_DIS
LIN {X 24.4632,Y 23.9512,Z 61,A 35.5498,B 24.8251,C -3.0507,E1 25.1174,E2 -312.5716} C_DIS
LIN {X 26.6225,Y 21.527,Z 61,A 30.9019,B 24.8252,C -3.049,E1 25.1258,E2 -307.9409} C_DIS
LIN {X 27.6419,Y 20.2012,Z 61,A 28.3944,B 24.8256,C -3.0463,E1 25.13,E2 -305.4391} C_DIS
LIN {X 28.5747,Y 18.8588,Z 61,A 25.4409,B 24.8267,C -3.0366,E1 25.1346,E2 -302.477} C_DIS
LIN {X 29.5164,Y 17.348,Z 61,A 22.5307,B 24.8274,C -3.0299,E1 25.1388,E2 -299.5658} C_DIS
LIN {X 30.2596,Y 16.0165,Z 61,A 20.1798,B 24.8279,C -3.0259,E1 25.142,E2 -297.2179} C_DIS
LIN {X 31.1082,Y 14.2985,Z 61,A 16.555,B 24.8296,C -3.0113,E1 25.1463,E2 -293.5779} C_DIS
LIN {X 32.0464,Y 12.0498,Z 61,A 12.3732,B 24.831,C -2.9983,E1 25.1506,E2 -289.3884} C_DIS
LIN {X 32.7002,Y 10.1421,Z 61,A 9.5852,B 24.8312,C -2.9968,E1 25.1531,E2 -286.6128} C_DIS
LIN {X 33.3069,Y 7.9274,Z 61,A 4.9109,B 24.8338,C -2.9735,E1 25.1563,E2 -281.9102} C_DIS
LIN {X 33.8016,Y 5.4436,Z 61,A 1.3333,B 24.8342,C -2.9701,E1 25.1581,E2 -278.3454} C_DIS
LIN {X 34.073,Y 3.3519,Z 61,A -2.5306,B 24.836,C -2.9544,E1 25.1593,E2 -274.4672} C_DIS
LIN {X 34.2255,Y 0.8907,Z 61,A -5.9936,B 24.8363,C -2.9511,E1 25.1598,E2 -271.0171} C_DIS
LIN {X 34.234,Y -0.4289,Z 61,A -8.6025,B 24.8377,C -2.9384,E1 25.1598,E2 -268.3936} C_DIS
LIN {X 34.1433,Y -2.5375,Z 61,A -11.9539,B 24.8387,C -2.9299,E1 25.1592,E2 -265.0421} C_DIS
LIN {X 33.9608,Y -4.339,Z 61,A -14.8256,B 24.8395,C -2.9228,E1 25.1583,E2 -262.1704} C_DIS
LIN {X 33.7229,Y -5.9122,Z 61,A -17.5477,B 24.8405,C -2.9136,E1 25.1571,E2 -259.4425} C_DIS
LIN {X 33.3312,Y -7.8235,Z 61,A -21.0107,B 24.8419,C -2.9006,E1 25.155,E2 -255.9689} C_DIS
LIN {X 32.7663,Y -9.9283,Z 61,A -24.7882,B 24.8433,C -2.8875,E1 25.1521,E2 -252.1821} C_DIS
LIN {X 31.9456,Y -12.3157,Z 61,A -28.6225,B 24.8441,C -2.8804,E1 25.1484,E2 -248.3524} C_DIS
LIN {X 31.3073,Y -13.8582,Z 61,A -32.1398,B 24.8461,C -2.8618,E1 25.1445,E2 -244.8103} C_DIS
LIN {X 29.6487,Y -17.1208,Z 61,A -37.2538,B 24.8465,C -2.8586,E1 25.1378,E2 -239.7157} C_DIS
LIN {X 28.2067,Y -19.4052,Z 61,A -43.1934,B 24.8499,C -2.8263,E1 25.1286,E2 -233.7292} C_DIS
LIN {X 25.2968,Y -23.0705,Z 61,A -50.9132,B 24.8519,C -2.8081,E1 25.1146,E2 -226.0015} C_DIS
LIN {X 23.1686,Y -25.2067,Z 61,A -55.4873,B 24.8524,C -2.8028,E1 25.1054,E2 -221.4337} C_DIS
LIN {X 20.6419,Y -27.3139,Z 61,A -59.9628,B 24.8522,C -2.805,E1 25.0957,E2 -216.9802} C_DIS
LIN {X 19.5642,Y -28.0964,Z 61,A -63.6273,B 24.8547,C -2.7815,E1 25.0872,E2 -213.2725} C_DIS
LIN {X 15.9335,Y -30.3033,Z 61,A -69.5799,B 24.8544,C -2.7841,E1 25.0729,E2 -207.3442} C_DIS
LIN {X 13.578,Y -31.4293,Z 61,A -74.5434,B 24.8559,C -2.7699,E1 25.0602,E2 -202.3594} C_DIS
LIN {X 11.1419,Y -32.3736,Z 61,A -78.4908,B 24.8559,C -2.7696,E1 25.0499,E2 -198.4196} C_DIS
LIN {X 9.0932,Y -33.0077,Z 61,A -82.0282,B 24.8563,C -2.7663,E1 25.0404,E2 -194.8805} C_DIS
LIN {X 6.6042,Y -33.5937,Z 61,A -86.8618,B 24.8574,C -2.7558,E1 25.0272,E2 -190.0281} C_DIS
LIN {X 3.6968,Y -34.037,Z 61,A -91.4663,B 24.8573,C -2.7565,E1 25.0144,E2 -185.429} C_DIS
LIN {X 1.0479,Y -34.2208,Z 61,A -94.973,B 24.8563,C -2.7658,E1 25.0047,E2 -181.9456} C_DIS
LIN {X 1.0479,Y -34.2208,Z 61,A -94.973,B 24.8563,C -2.7658,E1 25.0047,E2 -181.9456} C_DIS
Enddeposition()
LIN {X 0.2037,Y -33.2493,Z 61,A -96.7169,B 24.855,C -2.7787,E1 24.9999,E2 -180.2327} C_DIS
Startdeposition()
$VEL.CP = VEL_PRINT
LIN {X 1.2376,Y -33.2294,Z 61,A -93.5739,B 24.8533,C -2.7949,E1 25.0088,E2 -183.4137} C_DIS
LIN {X 3.4056,Y -33.077,Z 61,A -90.1141,B 24.8534,C -2.7934,E1 25.0184,E2 -186.8679} C_DIS
LIN {X 4.8616,Y -32.8939,Z 61,A -86.8624,B 24.8523,C -2.8038,E1 25.0275,E2 -190.1415} C_DIS
LIN {X 7.9397,Y -32.2901,Z 61,A -82.2136,B 24.8528,C -2.7993,E1 25.0401,E2 -194.7735} C_DIS
LIN {X 9.3148,Y -31.9202,Z 61,A -79.1754,B 24.8518,C -2.8092,E1 25.0483,E2 -197.8302} C_DIS
LIN {X 11.9154,Y -31.044,Z 61,A -74.5286,B 24.8512,C -2.8142,E1 25.0605,E2 -202.4792} C_DIS
LIN {X 14.4279,Y -29.9587,Z 61,A -70.3182,B 24.8512,C -2.8147,E1 25.0712,E2 -206.6804} C_DIS
LIN {X 15.7529,Y -29.2838,Z 61,A -67.2569,B 24.85,C -2.8255,E1 25.0788,E2 -209.7586} C_DIS
LIN {X 18.044,Y -27.9302,Z 61,A -63.0927,B 24.8497,C -2.8283,E1 25.0887,E2 -213.9164} C_DIS
LIN {X 19.5003,Y -26.9343,Z 61,A -59.2713,B 24.8479,C -2.8449,E1 25.0975,E2 -217.7638} C_DIS
LIN {X 22.3777,Y -24.5954,Z 61,A -53.5861,B 24.8475,C -2.8493,E1 25.1095,E2 -223.4374} C_DIS
LIN {X 24.4689,Y -22.5158,Z 61,A -47.8008,B 24.8451,C -2.8713,E1 25.1208,E2 -229.2498} C_DIS
LIN {X 26.1445,Y -20.5465,Z 61,A -44.3325,B 24.8454,C -2.8689,E1 25.1269,E2 -232.6964} C_DIS
LIN {X 27.4731,Y -18.733,Z 61,A -39.8056,B 24.8432,C -2.8885,E1 25.1342,E2 -237.2476} C_DIS
LIN {X 28.6335,Y -16.9058,Z 61,A -36.8933,B 24.8434,C -2.8873,E1 25.1384,E2 -240.1423} C_DIS
LIN {X 29.6848,Y -14.9835,Z 61,A -32.4106,B 24.8411,C -2.9082,E1 25.1443,E2 -244.6508} C_DIS
LIN {X 30.7611,Y -12.6274,Z 61,A -28.1849,B 24.84,C -2.918,E1 25.149,E2 -248.8766} C_DIS
LIN {X 31.5163,Y -10.6022,Z 61,A -24.7557,B 24.8392,C -2.925,E1 25.1522,E2 -252.3031} C_DIS
LIN {X 32.2558,Y -8.077,Z 61,A -19.3919,B 24.8364,C -2.9509,E1 25.1561,E2 -257.6975} C_DIS
LIN {X 32.7588,Y -5.708,Z 61,A -15.4347,B 24.8353,C -2.9608,E1 25.1581,E2 -261.6548} C_DIS
LIN {X 33.1404,Y -2.7208,Z 61,A -10.9844,B 24.8346,C -2.9663,E1 25.1594,E2 -266.0919} C_DIS
LIN {X 33.236,Y -1.0266,Z 61,A -7.9443,B 24.8334,C -2.9771,E1 25.1598,E2 -269.1396} C_DIS
LIN {X 33.249,Y 0.4639,Z 61,A -5.1262,B 24.8321,C -2.9888,E1 25.1597,E2 -271.9685} C_DIS
LIN {X 33.1166,Y 2.9963,Z 61,A -1.258,B 24.8314,C -2.9951,E1 25.1589,E2 -275.8287} C_DIS
LIN {X 32.9333,Y 4.5903,Z 61,A 1.6369,B 24.8302,C -3.0055,E1 25.1579,E2 -278.7311} C_DIS
LIN {X 32.6139,Y 6.483,Z 61,A 5.0853,B 24.8288,C -3.0175,E1 25.1561,E2 -282.1879} C_DIS
LIN {X 32.0855,Y 8.7298,Z 61,A 9.0488,B 24.8275,C -3.0292,E1 25.1534,E2 -286.1561} C_DIS
LIN {X 31.3718,Y 11.0224,Z 61,A 12.8387,B 24.8267,C -3.0363,E1 25.1501,E2 -289.9413} C_DIS
LIN {X 30.8266,Y 12.4666,Z 61,A 16.2464,B 24.8246,C -3.0544,E1 25.1466,E2 -293.3731} C_DIS
LIN {X 29.2927,Y 15.7366,Z 61,A 22.1381,B 24.8232,C -3.0665,E1 25.1392,E2 -299.2621} C_DIS
LIN {X 28.1253,Y 17.739,Z 61,A 25.6018,B 24.8229,C -3.0694,E1 25.1343,E2 -302.715} C_DIS
LIN {X 27.3144,Y 18.9633,Z 61,A 28.1231,B 24.8222,C -3.0756,E1 25.1303,E2 -305.2384} C_DIS
LIN {X 26.4116,Y 20.2021,Z 61,A 30.6224,B 24.8217,C -3.0799,E1 25.1261,E2 -307.7361} C_DIS
LIN {X 25.6694,Y 21.1374,Z 61,A 32.8856,B 24.8208,C -3.0875,E1 25.1221,E2 -310.0066} C_DIS
LIN {X 24.6533,Y 22.3144,Z 61,A 36.1277,B 24.8192,C -3.1009,E1 25.1161,E2 -313.2662} C_DIS
LIN {X 22.6607,Y 24.3353,Z 61,A 40.7673,B 24.8184,C -3.1075,E1 25.1068,E2 -317.902} C_DIS
LIN {X 20.6346,Y 26.0749,Z 61,A 44.6346,B 24.8186,C -3.1064,E1 25.0985,E2 -321.752} C_DIS
LIN {X 19.4266,Y 26.9873,Z 61,A 47.4239,B 24.8178,C -3.1132,E1 25.0923,E2 -324.5473} C_DIS
LIN {X 17.9952,Y 27.9618,Z 61,A 50.8871,B 24.8165,C -3.124,E1 25.0842,E2 -328.0246} C_DIS
LIN {X 16.3297,Y 28.9663,Z 61,A 54.089,B 24.8162,C -3.1268,E1 25.0764,E2 -331.2235} C_DIS
LIN {X 14.4707,Y 29.938,Z 61,A 57.5491,B 24.8159,C -3.1293,E1 25.0678,E2 -334.6801} C_DIS
LIN {X 13.1749,Y 30.5307,Z 61,A 60.3624,B 24.815,C -3.1363,E1 25.0606,E2 -337.5033} C_DIS
LIN {X 10.7733,Y 31.4586,Z 61,A 64.3098,B 24.8153,C -3.1344,E1 25.0503,E2 -341.4378} C_DIS
LIN {X 7.9038,Y 32.2989,Z 61,A 70.4406,B 24.8135,C -3.1492,E1 25.0337,E2 -347.5942} C_DIS
LIN {X 5.4519,Y 32.8019,Z 61,A 74.7552,B 24.8133,C -3.1507,E1 25.0218,E2 -351.9077} C_DIS
LIN {X 1.5203,Y 33.2172,Z 61,A 80.4232,B 24.8148,C -3.1383,E1 25.0062,E2 -357.543} C_DIS
LIN {X -0.415,Y 33.249,Z 61,A 84.2298,B 24.8143,C -3.1428,E1 24.9955,E2 -361.3602} C_DIS
LIN {X -2.5535,Y 33.1535,Z 61,A 87.9426,B 24.8144,C -3.1417,E1 24.9852,E2 -365.0714} C_DIS
LIN {X -4.4812,Y 32.9491,Z 61,A 91.0358,B 24.8149,C -3.1372,E1 24.9766,E2 -368.156} C_DIS
LIN {X -6.4567,Y 32.6188,Z 61,A 94.6399,B 24.8151,C -3.1362,E1 24.9667,E2 -371.7615} C_DIS
LIN {X -8.6986,Y 32.0939,Z 61,A 99.0304,B 24.8151,C -3.1367,E1 24.9548,E2 -376.1596} C_DIS
LIN {X -10.7999,Y 31.4497,Z 61,A 103.3349,B 24.8149,C -3.1374,E1 24.9434,E2 -380.4739} C_DIS
LIN {X -14.5367,Y 29.9059,Z 61,A 109.0864,B 24.8175,C -3.1156,E1 24.9288,E2 -386.1869} C_DIS
LIN {X -15.7389,Y 29.2915,Z 61,A 111.7148,B 24.8176,C -3.1147,E1 24.9223,E2 -388.8203} C_DIS
LIN {X -17.455,Y 28.3018,Z 61,A 115.1553,B 24.8183,C -3.1089,E1 24.914,E2 -392.2576} C_DIS
LIN {X -20.0805,Y 26.5037,Z 61,A 121.8695,B 24.8183,C -3.1094,E1 24.8988,E2 -398.9964} C_DIS
LIN {X -22.4879,Y 24.4937,Z 61,A 126.2015,B 24.8208,C -3.0877,E1 24.8898,E2 -403.2937} C_DIS
LIN {X -24.0316,Y 22.9814,Z 61,A 129.7609,B 24.8219,C -3.0775,E1 24.8828,E2 -406.8439} C_DIS
LIN {X -25.455,Y 21.3953,Z 61,A 134.7361,B 24.8217,C -3.0797,E1 24.8738,E2 -411.847} C_DIS
LIN {X -28.0868,Y 17.7997,Z 61,A 141.0367,B 24.8254,C -3.0473,E1 24.8638,E2 -418.1011} C_DIS
LIN {X -28.8825,Y 16.4764,Z 61,A 143.7677,B 24.8262,C -3.0405,E1 24.86,E2 -420.8299} C_DIS
LIN {X -29.6814,Y 14.9899,Z 61,A 146.925,B 24.8269,C -3.0342,E1 24.8559,E2 -423.9891} C_DIS
LIN {X -30.8384,Y 12.4374,Z 61,A 152.4416,B 24.8279,C -3.0257,E1 24.8498,E2 -429.5157} C_DIS
LIN {X -31.7392,Y 9.9153,Z 61,A 156.8485,B 24.8297,C -3.01,E1 24.846,E2 -433.9102} C_DIS
LIN {X -32.457,Y 7.2278,Z 61,A 161.5167,B 24.8315,C -2.9942,E1 24.8429,E2 -438.5679} C_DIS
LIN {X -32.9745,Y 4.2859,Z 61,A 166.9535,B 24.833,C -2.9805,E1 24.8406,E2 -444.0043} C_DIS
LIN {X -33.2243,Y 1.3544,Z 61,A 171.6066,B 24.8352,C -2.9612,E1 24.8398,E2 -448.6393} C_DIS
LIN {X -33.2386,Y -0.9421,Z 61,A 174.975,B 24.8371,C -2.9442,E1 24.8398,E2 -451.9871} C_DIS
LIN {X -33.1591,Y -2.4833,Z 61,A 178.2097,B 24.8375,C -2.9405,E1 24.8404,E2 -455.2326} C_DIS
LIN {X -32.953,Y -4.4518,Z 61,A -178.5433,B 24.8388,C -2.9287,E1 24.8415,E2 -458.4707} C_DIS
LIN {X -32.6837,Y -6.1197,Z 61,A -175.7859,B 24.8399,C -2.9186,E1 24.8428,E2 -461.2204} C_DIS
LIN {X -32.4295,Y -7.3508,Z 61,A -173.1835,B 24.8403,C -2.9157,E1 24.8444,E2 -463.831} C_DIS
LIN {X -31.8574,Y -9.5287,Z 61,A -169.7396,B 24.8419,C -2.9006,E1 24.8469,E2 -467.2589} C_DIS
LIN {X -31.5023,Y -10.6437,Z 61,A -166.9912,B 24.8419,C -2.9009,E1 24.8494,E2 -470.0236} C_DIS
LIN {X -30.5236,Y -13.1911,Z 61,A -162.5281,B 24.8435,C -2.8856,E1 24.8541,E2 -474.475} C_DIS
LIN {X -29.5038,Y -15.3377,Z 61,A -159.0137,B 24.8453,C -2.8696,E1 24.8584,E2 -477.9701} C_DIS
LIN {X -28.8549,Y -16.5252,Z 61,A -156.0209,B 24.8453,C -2.8692,E1 24.8625,E2 -480.9775} C_DIS
LIN {X -27.6567,Y -18.461,Z 61,A -152.4369,B 24.8467,C -2.8564,E1 24.8678,E2 -484.5491} C_DIS
LIN {X -26.887,Y -19.5649,Z 61,A -149.9283,B 24.8471,C -2.8524,E1 24.8719,E2 -487.0605} C_DIS
LIN {X -25.7967,Y -20.9814,Z 61,A -146.8681,B 24.8479,C -2.8451,E1 24.8772,E2 -490.1176} C_DIS
LIN {X -24.6404,Y -22.3288,Z 61,A -143.7263,B 24.8486,C -2.8392,E1 24.883,E2 -493.2592} C_DIS
LIN {X -23.3559,Y -23.668,Z 61,A -140.6226,B 24.8494,C -2.8317,E1 24.8891,E2 -496.3583} C_DIS
LIN {X -22.136,Y -24.813,Z 61,A -137.5892,B 24.8498,C -2.8275,E1 24.8954,E2 -499.3939} C_DIS
LIN {X -20.5798,Y -26.118,Z 61,A -134.3283,B 24.8507,C -2.8189,E1 24.9024,E2 -502.6467} C_DIS
LIN {X -19.3641,Y -27.0318,Z 61,A -131.8535,B 24.8513,C -2.8131,E1 24.9079,E2 -505.1165} C_DIS
LIN {X -18.2498,Y -27.7963,Z 61,A -129.2905,B 24.8515,C -2.8118,E1 24.9139,E2 -507.6848} C_DIS
LIN {X -16.9366,Y -28.6154,Z 61,A -126.6679,B 24.8519,C -2.8075,E1 24.9202,E2 -510.3053} C_DIS
LIN {X -14.8115,Y -29.7709,Z 61,A -121.5179,B 24.8514,C -2.8123,E1 24.933,E2 -515.4807} C_DIS
LIN {X -12.9589,Y -30.6228,Z 61,A -117.8052,B 24.8516,C -2.8108,E1 24.9425,E2 -519.1985} C_DIS
LIN {X -9.2656,Y -31.9354,Z 61,A -111.9897,B 24.8532,C -2.7956,E1 24.9579,E2 -524.9885} C_DIS
LIN {X -6.793,Y -32.5508,Z 61,A -106.9954,B 24.8527,C -2.8001,E1 24.9715,E2 -530} C_DIS
LIN {X -4.8126,Y -32.902,Z 61,A -104.0453,B 24.8534,C -2.7935,E1 24.9796,E2 -532.9369} C_DIS
LIN {X -3.194,Y -33.0981,Z 61,A -101.4811,B 24.8537,C -2.7904,E1 24.9867,E2 -535.4954} C_DIS
LIN {X -1.6187,Y -33.2129,Z 61,A -98.4576,B 24.8534,C -2.794,E1 24.9952,E2 -538.5282} C_DIS
LIN {X 0.2037,Y -33.2493,Z 61,A -96.7167,B 24.855,C -2.7786,E1 25,E2 -540.2327} C_DIS
Enddeposition()
LIN {X 0.2037,Y -33.2493,Z 61,A -96.7167,B 24.855,C -2.7786,E1 25,E2 -540.2327} C_DIS
Startdeposition()
$VEL.CP = VEL_PRINT
LIN {X -0.5474,Y -32.2622,Z 61,A -98.3768,B 24.8536,C -2.7919,E1 24.9954,E2 -538.6042} C_DIS
LIN {X -2.6629,Y -32.1566,Z 61,A -102.7647,B 24.8543,C -2.7852,E1 24.9831,E2 -534.1987} C_DIS
LIN {X -5.7647,Y -31.7478,Z 61,A -108.1222,B 24.8539,C -2.7887,E1 24.9684,E2 -528.8447} C_DIS
LIN {X -7.6494,Y -31.3469,Z 61,A -111.1628,B 24.8533,C -2.7942,E1 24.9601,E2 -525.8133} C_DIS
LIN {X -10.469,Y -30.5214,Z 61,A -117.1892,B 24.8538,C -2.79,E1 24.944,E2 -519.7662} C_DIS
LIN {X -13.1387,Y -29.4706,Z 61,A -121.9435,B 24.8529,C -2.7984,E1 24.9318,E2 -515.021} C_DIS
LIN {X -15.5816,Y -28.2558,Z 61,A -126.6591,B 24.8521,C -2.8057,E1 24.9202,E2 -510.3097} C_DIS
LIN {X -17.8707,Y -26.8657,Z 61,A -131.1185,B 24.8511,C -2.8154,E1 24.9097,E2 -505.8594} C_DIS
LIN {X -19.2091,Y -25.9264,Z 61,A -134.5803,B 24.8511,C -2.8153,E1 24.9018,E2 -502.385} C_DIS
LIN {X -21.4335,Y -24.1199,Z 61,A -139.3181,B 24.8498,C -2.8277,E1 24.8917,E2 -497.6587} C_DIS
LIN {X -23.125,Y -22.5023,Z 61,A -142.9768,B 24.8484,C -2.8404,E1 24.8845,E2 -494.0151} C_DIS
LIN {X -23.9384,Y -21.6362,Z 61,A -145.6511,B 24.8484,C -2.8402,E1 24.8794,E2 -491.3284} C_DIS
LIN {X -25.4335,Y -19.8573,Z 61,A -149.8769,B 24.8475,C -2.8488,E1 24.872,E2 -487.1035} C_DIS
LIN {X -26.5961,Y -18.2708,Z 61,A -153.4537,B 24.8467,C -2.8566,E1 24.8663,E2 -483.5278} C_DIS
LIN {X -28.0311,Y -15.9818,Z 61,A -157.4896,B 24.8447,C -2.875,E1 24.8604,E2 -479.5152} C_DIS
LIN {X -29.0945,Y -13.9521,Z 61,A -162.6609,B 24.8445,C -2.8773,E1 24.8539,E2 -474.3215} C_DIS
LIN {X -30.0741,Y -11.6924,Z 61,A -166.396,B 24.8426,C -2.8945,E1 24.85,E2 -470.6068} C_DIS
LIN {X -30.735,Y -9.8245,Z 61,A -170.1652,B 24.8417,C -2.9027,E1 24.8466,E2 -466.8358} C_DIS
LIN {X -31.2532,Y -8.0241,Z 61,A -173.2509,B 24.8404,C -2.9144,E1 24.8443,E2 -463.7602} C_DIS
LIN {X -31.6367,Y -6.3472,Z 61,A -176.5037,B 24.8396,C -2.9221,E1 24.8424,E2 -460.5066} C_DIS
LIN {X -31.9775,Y -4.3148,Z 61,A -179.8739,B 24.8381,C -2.9354,E1 24.841,E2 -457.1483} C_DIS
LIN {X -32.1461,Y -2.7892,Z 61,A 177.3143,B 24.8372,C -2.9432,E1 24.8402,E2 -454.3382} C_DIS
LIN {X -32.251,Y -1.0105,Z 61,A 173.8229,B 24.8364,C -2.9506,E1 24.8398,E2 -450.8435} C_DIS
LIN {X -32.2581,Y 0.7696,Z 61,A 170.926,B 24.8351,C -2.9624,E1 24.8398,E2 -447.9575} C_DIS
LIN {X -32.1752,Y 2.4336,Z 61,A 167.7621,B 24.8342,C -2.9702,E1 24.8404,E2 -444.7931} C_DIS
LIN {X -31.9605,Y 4.4365,Z 61,A 164.0913,B 24.833,C -2.9806,E1 24.8417,E2 -441.1254} C_DIS
LIN {X -31.6122,Y 6.4669,Z 61,A 160.5011,B 24.8317,C -2.9925,E1 24.8435,E2 -437.5423} C_DIS
LIN {X -31.1898,Y 8.2682,Z 61,A 157.1888,B 24.8306,C -3.0024,E1 24.8458,E2 -434.2344} C_DIS
LIN {X -30.7384,Y 9.8139,Z 61,A 154.5647,B 24.8294,C -3.0129,E1 24.8479,E2 -431.6202} C_DIS
LIN {X -30.1797,Y 11.4164,Z 61,A 151.2018,B 24.8287,C -3.0193,E1 24.8511,E2 -428.2537} C_DIS
LIN {X -29.5143,Y 13.041,Z 61,A 148.2213,B 24.8275,C -3.0295,E1 24.8544,E2 -425.2811} C_DIS
LIN {X -28.6337,Y 14.8742,Z 61,A 143.8532,B 24.8269,C -3.0342,E1 24.8599,E2 -420.9008} C_DIS
LIN {X -27.0419,Y 17.6042,Z 61,A 138.4246,B 24.825,C -3.0511,E1 24.8678,E2 -415.4849} C_DIS
LIN {X -25.3117,Y 20.0117,Z 61,A 133.6608,B 24.823,C -3.0688,E1 24.8757,E2 -410.7406} C_DIS
LIN {X -24.2704,Y 21.2627,Z 61,A 130.0008,B 24.8228,C -3.0699,E1 24.8824,E2 -407.0665} C_DIS
LIN {X -21.8103,Y 23.7794,Z 61,A 124.2249,B 24.8207,C -3.0882,E1 24.8939,E2 -401.3104} C_DIS
LIN {X -20.7161,Y 24.7387,Z 61,A 121.083,B 24.8206,C -3.0892,E1 24.9006,E2 -398.1587} C_DIS
LIN {X -18.1357,Y 26.688,Z 61,A 115.7631,B 24.8188,C -3.1041,E1 24.9126,E2 -392.856} C_DIS
LIN {X -15.9646,Y 28.0409,Z 61,A 111.2926,B 24.8178,C -3.1128,E1 24.9233,E2 -388.3925} C_DIS
LIN {X -14.3578,Y 28.8964,Z 61,A 107.7812,B 24.8175,C -3.1155,E1 24.9321,E2 -384.878} C_DIS
LIN {X -11.7963,Y 30.0329,Z 61,A 103.6271,B 24.8158,C -3.1299,E1 24.9427,E2 -380.7488} C_DIS
LIN {X -10.3847,Y 30.5502,Z 61,A 101.0677,B 24.8153,C -3.1343,E1 24.9494,E2 -378.1947} C_DIS
LIN {X -8.7834,Y 31.0482,Z 61,A 97.3578,B 24.8157,C -3.1306,E1 24.9593,E2 -374.4696} C_DIS
LIN {X -6.4188,Y 31.6218,Z 61,A 92.4968,B 24.8159,C -3.1291,E1 24.9726,E2 -369.5992} C_DIS
LIN {X -2.9881,Y 32.1281,Z 61,A 86.7854,B 24.815,C -3.1371,E1 24.9884,E2 -363.9027} C_DIS
LIN {X -0.6867,Y 32.2593,Z 61,A 82.6874,B 24.8148,C -3.1383,E1 24.9998,E2 -359.8069} C_DIS
LIN {X 1.3718,Y 32.2377,Z 61,A 78.4715,B 24.8155,C -3.1328,E1 25.0116,E2 -355.579} C_DIS
LIN {X 5.1633,Y 31.8512,Z 61,A 72.8802,B 24.8141,C -3.1442,E1 25.027,E2 -350.0188} C_DIS
LIN {X 7.4939,Y 31.3849,Z 61,A 67.5295,B 24.8158,C -3.1297,E1 25.0417,E2 -344.6409} C_DIS
LIN {X 10.1053,Y 30.644,Z 61,A 63.5243,B 24.8152,C -3.1354,E1 25.0523,E2 -340.6563} C_DIS
LIN {X 11.792,Y 30.0348,Z 61,A 60.2844,B 24.8156,C -3.1318,E1 25.0608,E2 -337.4148} C_DIS
LIN {X 13.8956,Y 29.1216,Z 61,A 56.2619,B 24.816,C -3.1279,E1 25.0711,E2 -333.3929} C_DIS
LIN {X 15.2278,Y 28.4476,Z 61,A 53.4394,B 24.8167,C -3.1225,E1 25.078,E2 -330.5655} C_DIS
LIN {X 16.9202,Y 27.4747,Z 61,A 50.3263,B 24.8167,C -3.1218,E1 25.0855,E2 -327.4604} C_DIS
LIN {X 18.3815,Y 26.5193,Z 61,A 46.9844,B 24.8177,C -3.1139,E1 25.0933,E2 -324.1111} C_DIS
LIN {X 19.8283,Y 25.4561,Z 61,A 43.9888,B 24.8181,C -3.1108,E1 25.0999,E2 -321.1188} C_DIS
LIN {X 21.2194,Y 24.3081,Z 61,A 40.672,B 24.8189,C -3.1034,E1 25.107,E2 -317.7973} C_DIS
Enddeposition()
END
